	sDate := WORD_TO_STRING(TimeStruct.wYear);
	sDate := CONCAT(sDate,'-');
	IF TimeStruct.wMonth < 10 THEN sDate := CONCAT(sDate, '0');	END_IF
	sDate := CONCAT(sDate,WORD_TO_STRING(TimeStruct.wMonth));
	sDate := CONCAT(sDate,'-');
	IF TimeStruct.wDay < 10 THEN sDate := CONCAT(sDate, '0');	END_IF
	sDate := CONCAT(sDate,WORD_TO_STRING(TimeStruct.wDay));
	
	sTime := '';
	IF TimeStruct.wHour < 10 THEN sTime := CONCAT(sTime, '0');	END_IF
	sTime := CONCAT(sTime, WORD_TO_STRING(TimeStruct.wHour));
	sTime := CONCAT(sTime,':');
	IF TimeStruct.wMinute < 10 THEN sTime := CONCAT(sTime, '0');END_IF
	sTime := CONCAT(sTime,WORD_TO_STRING(TimeStruct.wMinute));
	sTime := CONCAT(sTime,':');
	IF TimeStruct.wSecond < 10 THEN sTime := CONCAT(sTime, '0');END_IF
	sTime := CONCAT(sTime,WORD_TO_STRING(TimeStruct.wSecond)); 
	sTime := CONCAT(sTime,'.');
	IF TimeStruct.wMilliseconds < 100 THEN sTime := CONCAT(sTime, '0');END_IF
	IF TimeStruct.wMilliseconds <  10 THEN sTime := CONCAT(sTime, '0');END_IF
	sTime := CONCAT(sTime,WORD_TO_STRING(TimeStruct.wMilliseconds)); 




IF NOT ((stCommand.eCommandType = eMoverCommand_eGearOutOfSync) OR (stCommand.eCommandType = eMoverCommand_eGearInInSync)) THEN
	THIS^.stLastCommand := stCommand;
END_IF



stMoverAxisCommand := stMoverAxisCommandClear;
CASE _eLogSeverity OF
	
	TcEventSeverity.Critical :;
	
	TcEventSeverity.ERROR:;
	
	TcEventSeverity.INFO:;
	
	TcEventSeverity.VERBOSE:
		
		CASE stCommand.eCommandType OF	

		eMoverCommand_eSetPosition:
			fbFormatString.sFormat := 'SetPosition: X:%.1f;Y:%.1f;C:%.1f';
			fbFormatString.arg1    := F_LREAL(stCommand.stSetPosition.fPositionX);
			fbFormatString.arg2    := F_LREAL(stCommand.stSetPosition.fPositionY);
			fbFormatString.arg3    := F_LREAL(stCommand.stSetPosition.fPositionC);		
			fbFormatString();				
			stMoverAxisCommand.sCommandType   := MoverCommandToString(stCommand.eCommandType);
			stMoverAxisCommand.sTimeStamp 	  := stCommand.stTimeStamp;
			stMoverAxisCommand.sTimeStampDate := sDate;
			stMoverAxisCommand.sTimeStampTime := sTime;
			stMoverAxisCommand.sStation       := stCommand.sText;
			stMoverAxisCommand.sText      	  := fbFormatString.sOut;
				
		eMoverCommand_eReset:
			stMoverAxisCommand.sCommandType   := MoverCommandToString(stCommand.eCommandType);
			stMoverAxisCommand.sTimeStamp 	  := stCommand.stTimeStamp;
			stMoverAxisCommand.sTimeStampDate := sDate;
			stMoverAxisCommand.sTimeStampTime := sTime;
			stMoverAxisCommand.sStation       := stCommand.sText;
			stMoverAxisCommand.sText      	  := 'Reset Cmd';		
	
		eMoverCommand_eEnable:
			stMoverAxisCommand.sCommandType   := MoverCommandToString(stCommand.eCommandType);
			stMoverAxisCommand.sTimeStamp 	  := stCommand.stTimeStamp;
			stMoverAxisCommand.sTimeStampDate := sDate;
			stMoverAxisCommand.sTimeStampTime := sTime;
			stMoverAxisCommand.sStation       := stCommand.sText;
			stMoverAxisCommand.sText      	  := 'Enable Cmd';

		eMoverCommand_eDisable:			
			stMoverAxisCommand.sCommandType   := MoverCommandToString(stCommand.eCommandType);
			stMoverAxisCommand.sStation       := stCommand.sStation;
			stMoverAxisCommand.sText          := 'Disable Cmd';
			stMoverAxisCommand.sTimeStamp 	  := stCommand.stTimeStamp;
			stMoverAxisCommand.sTimeStampDate := sDate;
			stMoverAxisCommand.sTimeStampTime := sTime;

		eMoverCommand_eMoveToPosition:
			fbFormatString.sFormat := 'TargetPos: X:%.1f;Y:%.1f;C:%.1f;Velo:%.2f;Acc:%.0f;Dec:%.0f;Jerk:%.0f';
			fbFormatString.arg1    := F_LREAL(stCommand.stMoveToPositionXYC.fTargetPositionX);
			fbFormatString.arg2    := F_LREAL(stCommand.stMoveToPositionXYC.fTargetPositionY);
			fbFormatString.arg3    := F_LREAL(stCommand.stMoveToPositionXYC.fTargetPositionC);	
			fbFormatString.arg4    := F_LREAL(stCommand.stMoveToPositionXYC.fVelo );	
			fbFormatString.arg5    := F_LREAL(stCommand.stMoveToPositionXYC.fAcc );	
			fbFormatString.arg6    := F_LREAL(stCommand.stMoveToPositionXYC.fDec );
			fbFormatString.arg7    := F_LREAL(stCommand.stMoveToPositionXYC.fJerk );	
			fbFormatString();		
			stMoverAxisCommand.sCommandType   := MoverCommandToString(stCommand.eCommandType);
			stMoverAxisCommand.sStation       := stCommand.sText;	
			stMoverAxisCommand.sText          := fbFormatString.sOut;
			stMoverAxisCommand.sTimeStamp     := stCommand.stTimeStamp;
			stMoverAxisCommand.sTimeStampDate := sDate;
			stMoverAxisCommand.sTimeStampTime := sTime;			

		eMoverCommand_eMoveToPositionXYC:
			fbFormatString.sFormat := 'TargetPos: X:%.1f;Y:%.1f;C:%.1f;Velo:%.2f;Acc:%.0f;Dec:%.0f;Jerk:%.0f';
			fbFormatString.arg1    := F_LREAL(stCommand.stMoveToPositionXYC.fTargetPositionX);
			fbFormatString.arg2    := F_LREAL(stCommand.stMoveToPositionXYC.fTargetPositionY);
			fbFormatString.arg3    := F_LREAL(stCommand.stMoveToPositionXYC.fTargetPositionC);	
			fbFormatString.arg4    := F_LREAL(stCommand.stMoveToPositionXYC.fVelo );	
			fbFormatString.arg5    := F_LREAL(stCommand.stMoveToPositionXYC.fAcc );	
			fbFormatString.arg6    := F_LREAL(stCommand.stMoveToPositionXYC.fDec );
			fbFormatString.arg7    := F_LREAL(stCommand.stMoveToPositionXYC.fJerk );	
			fbFormatString();		
			stMoverAxisCommand.sCommandType   := MoverCommandToString(stCommand.eCommandType);
			stMoverAxisCommand.sStation       := stCommand.sText;	
			stMoverAxisCommand.sText          := fbFormatString.sOut;
			stMoverAxisCommand.sTimeStamp     := stCommand.stTimeStamp;
			stMoverAxisCommand.sTimeStampDate := sDate;
			stMoverAxisCommand.sTimeStampTime := sTime;	

		eMoverCommand_eMoveToPositionExt:
			fbFormatString.sFormat := 'XargetPos: X:%.1f;Y:%.1f;C:%.1f;V:%.2f;A:%.0f;D:%.0f;J:%.0f';
			fbFormatString.arg1    := F_LREAL(stCommand.stMoveToPositionExt.fTargetPositionX);
			fbFormatString.arg2    := F_LREAL(stCommand.stMoveToPositionExt.fTargetPositionY);
			fbFormatString.arg3    := F_LREAL(stCommand.stMoveToPositionExt.fTargetPositionC);	
			fbFormatString.arg4    := F_LREAL(stCommand.stMoveToPositionExt.fVelo );	
			fbFormatString.arg5    := F_LREAL(stCommand.stMoveToPositionExt.fAcc );	
			fbFormatString.arg6    := F_LREAL(stCommand.stMoveToPositionExt.fDec );
			fbFormatString.arg7    := F_LREAL(stCommand.stMoveToPositionExt.fJerk );	
			
			fbFormatString();	
			tempString06 := fbFormatString.sOut;			
			IF stCommand.stMoveToPositionExt.stMoveToPositionOptions.useOrientation THEN
				tempString06 := CONCAT(tempString06,' Or:T');
			ELSE
				tempString06 := CONCAT(tempString06,' Or:F');
			END_IF
					
				
			stMoverAxisCommand.sCommandType   := MoverCommandToString(stCommand.eCommandType);
			stMoverAxisCommand.sStation       := stCommand.sText;	
			stMoverAxisCommand.sText          := tempString06;
			stMoverAxisCommand.sTimeStamp     := stCommand.stTimeStamp;
			stMoverAxisCommand.sTimeStampDate := sDate;
			stMoverAxisCommand.sTimeStampTime := sTime;	


			
		eMoverCommand_eMoveA:
			stMoverAxisCommand.sCommandType   := MoverCommandToString(stCommand.eCommandType);
			stMoverAxisCommand.sStation 	  := stCommand.sStation;
			fbFormatString.sFormat	 		  := 'Position: %.2f; Vel %.0f; acc %.0f; Dec %.0f; Jerk %.0f;   '; 
			fbFormatString.arg1 			  := F_LREAL(stCommand.stMoveOnTrackParameter.fTargetPosition);
			fbFormatString.arg2 			  := F_LREAL(stCommand.stMoveOnTrackParameter.fVelo);
			fbFormatString.arg3 			  := F_LREAL(stCommand.stMoveOnTrackParameter.fAcc);
			fbFormatString.arg4 			  := F_LREAL(stCommand.stMoveOnTrackParameter.fDec);
			fbFormatString.arg5 			  := F_LREAL(stCommand.stMoveOnTrackParameter.fJerk);
			fbFormatString();
			stMoverAxisCommand.sText 		  := fbFormatString.sOut;
			stMoverAxisCommand.sTimeStamp 	  := stCommand.stTimeStamp;
			stMoverAxisCommand.sTimeStampDate := sDate;
			stMoverAxisCommand.sTimeStampTime := sTime;	
	
		eMoverCommand_eMoveB:
			stMoverAxisCommand.sCommandType   := MoverCommandToString(stCommand.eCommandType);
			stMoverAxisCommand.sStation 	  := stCommand.sStation;
			fbFormatString.sFormat	 		  := 'Position: %.2f; Vel %.0f; acc %.0f; Dec %.0f; Jerk %.0f;   '; 
			fbFormatString.arg1 			  := F_LREAL(stCommand.stMoveOnTrackParameter.fTargetPosition);
			fbFormatString.arg2 			  := F_LREAL(stCommand.stMoveOnTrackParameter.fVelo);
			fbFormatString.arg3 			  := F_LREAL(stCommand.stMoveOnTrackParameter.fAcc);
			fbFormatString.arg4 			  := F_LREAL(stCommand.stMoveOnTrackParameter.fDec);
			fbFormatString.arg5 			  := F_LREAL(stCommand.stMoveOnTrackParameter.fJerk);
			fbFormatString();
			stMoverAxisCommand.sText 		  := fbFormatString.sOut;
			stMoverAxisCommand.sTimeStamp 	  := stCommand.stTimeStamp;
			stMoverAxisCommand.sTimeStampDate := sDate;
			stMoverAxisCommand.sTimeStampTime := sTime;	

		eMoverCommand_eMoveC:
			stMoverAxisCommand.sCommandType   := MoverCommandToString(stCommand.eCommandType);
			stMoverAxisCommand.sStation 	  := stCommand.sStation;
			fbFormatString.sFormat	 		  := 'Position: %.2f; Vel %.0f; acc %.0f; Dec %.0f; Jerk %.0f;   '; 
			fbFormatString.arg1 			  := F_LREAL(stCommand.stMoveOnTrackParameter.fTargetPosition);
			fbFormatString.arg2 			  := F_LREAL(stCommand.stMoveOnTrackParameter.fVelo);
			fbFormatString.arg3 			  := F_LREAL(stCommand.stMoveOnTrackParameter.fAcc);
			fbFormatString.arg4 			  := F_LREAL(stCommand.stMoveOnTrackParameter.fDec);
			fbFormatString.arg5 			  := F_LREAL(stCommand.stMoveOnTrackParameter.fJerk);
			fbFormatString();
			stMoverAxisCommand.sText 		  := fbFormatString.sOut;
			stMoverAxisCommand.sTimeStamp 	  := stCommand.stTimeStamp;
			stMoverAxisCommand.sTimeStampDate := sDate;
			stMoverAxisCommand.sTimeStampTime := sTime;				
					
		eMoverCommand_eMoveZ:
			stMoverAxisCommand.sCommandType   := MoverCommandToString(stCommand.eCommandType);
			fbFormatString.sFormat	 		  := 'Position: %.2f; Vel %.0f; acc %.0f; Dec %.0f; Jerk %.0f;   '; 
			fbFormatString.arg1 			  := F_LREAL(stCommand.stMoveOnTrackParameter.fTargetPosition);
			fbFormatString.arg2 			  := F_LREAL(stCommand.stMoveOnTrackParameter.fVelo);
			fbFormatString.arg3 			  := F_LREAL(stCommand.stMoveOnTrackParameter.fAcc);
			fbFormatString.arg4 			  := F_LREAL(stCommand.stMoveOnTrackParameter.fDec);
			fbFormatString.arg5 			  := F_LREAL(stCommand.stMoveOnTrackParameter.fJerk);
			fbFormatString();
			stMoverAxisCommand.sText 		  := fbFormatString.sOut;
			stMoverAxisCommand.sStation 	  := stCommand.sStation;
			stMoverAxisCommand.sTimeStamp 	  := stCommand.stTimeStamp;
			stMoverAxisCommand.sTimeStampDate := sDate;
			stMoverAxisCommand.sTimeStampTime := sTime;	
			
		eMoverCommand_eJoinTrack:
			stMoverAxisCommand.sCommandType   := MoverCommandToString(stCommand.eCommandType);
			fbFormatString.sFormat            := 'TrackOID: %d; Vel %.0f; acc %.0f; Jerk %.0f; ';
			fbFormatString.arg1               := F_UDINT(stCommand.stJoinTrackParameter.nTargetTrack);
			fbFormatString.arg2				  := F_LREAL(stCommand.stJoinTrackParameter.fVelo); 
			fbFormatString.arg3				  := F_LREAL(stCommand.stJoinTrackParameter.fAcc); 
			fbFormatString.arg4				  := F_LREAL(stCommand.stJoinTrackParameter.fJerk); 
			fbFormatString();
			stMoverAxisCommand.sText          := fbFormatString.sOut;	
			stMoverAxisCommand.sStation 	  := stCommand.sStation;
			stMoverAxisCommand.sTimeStamp 	  := stCommand.stTimeStamp;		
			stMoverAxisCommand.sTimeStampDate := sDate;
			stMoverAxisCommand.sTimeStampTime := sTime;			
			
		eMoverCommand_eLeaveTrack:
			stMoverAxisCommand.sCommandType   := MoverCommandToString(stCommand.eCommandType);
			fbFormatString.sFormat            := 'Pos: X:%.1f; Y:%.1f; C:%.1f; Vel:%.0f  Acc:%.0f; Dec:%.0f Jerk %.0f';
			fbFormatString.arg1               := F_LREAL(stCommand.stLeaveTrackParameter.fPositionX);
			fbFormatString.arg2               := F_LREAL(stCommand.stLeaveTrackParameter.fPositionY);
			fbFormatString.arg3               := F_LREAL(stCommand.stLeaveTrackParameter.fPositionC);
			fbFormatString.arg4				  := F_LREAL(stCommand.stLeaveTrackParameter.fVelo); 
			fbFormatString.arg5				  := F_LREAL(stCommand.stLeaveTrackParameter.fAcc); 
			fbFormatString.arg6				  := F_LREAL(stCommand.stLeaveTrackParameter.fDec); 
			fbFormatString.arg7				  := F_LREAL(stCommand.stLeaveTrackParameter.fJerk); 
			fbFormatString();
			stMoverAxisCommand.sText          := fbFormatString.sOut;	
			stMoverAxisCommand.sStation 	  := stCommand.sStation;
			stMoverAxisCommand.sTimeStamp 	  := stCommand.stTimeStamp;		
			stMoverAxisCommand.sTimeStampDate := sDate;
			stMoverAxisCommand.sTimeStampTime := sTime;			
	

		eMoverCommand_eLeaveTrackInPosition:
			stMoverAxisCommand.sCommandType   := MoverCommandToString(stCommand.eCommandType);
			fbFormatString.sFormat            := 'Pos: X:%.1f; Y:%.1f; C:%.1f';
			fbFormatString.arg1               := F_LREAL(stCommand.stLeaveTrackInPositionParameter.fPositionX);
			fbFormatString.arg2               := F_LREAL(stCommand.stLeaveTrackInPositionParameter.fPositionY);
			fbFormatString.arg3               := F_LREAL(stCommand.stLeaveTrackInPositionParameter.fPositionC);
			fbFormatString();
			stMoverAxisCommand.sText          := fbFormatString.sOut;	
			stMoverAxisCommand.sStation 	  := stCommand.sStation;
			stMoverAxisCommand.sTimeStamp 	  := stCommand.stTimeStamp;		
			stMoverAxisCommand.sTimeStampDate := sDate;
			stMoverAxisCommand.sTimeStampTime := sTime;			

		eMoverCommand_eMoveModOnTrack:
			fbFormatString.sFormat := 'TargetPos:%.4f;Velo:%.2f;Acc:%.0f;Jerk:%.0f;Gap:%.0f;TargetTrack:%d $n ;ActSetPos:%.2f;ActSetOid:%d;ActVelo:%.0f;ActAcc:%.0f;';
			fbFormatString.arg1 := F_LREAL(stCommand.stMoveOnTrackParameter.fTargetPosition);
			fbFormatString.arg2 := F_LREAL(stCommand.stMoveOnTrackParameter.fVelo );	
			fbFormatString.arg3 := F_LREAL(stCommand.stMoveOnTrackParameter.fAcc );	
			fbFormatString.arg4 := F_LREAL(stCommand.stMoveOnTrackParameter.fJerk );
			fbFormatString.arg5 := F_LREAL(stCommand.stMoveOnTrackParameter.fGap);
			fbFormatString.arg6 := F_UDINT(stCommand.stMoveOnTrackParameter.nTargetTrackOid);
			fbFormatString.arg7 := F_LREAL(stCommand.stActualParameter.fSetTrackPosition);
			fbFormatString.arg8 := F_UDINT(stCommand.stActualParameter.nTrackOid);	
			fbFormatString.arg9 := F_LREAL(stCommand.stActualParameter.fSetVelo);	
			fbFormatString.arg10:= F_LREAL(stCommand.stActualParameter.fSetAcc);			
			fbFormatString();
			
			stMoverAxisCommand.sCommandType   := MoverCommandToString(stCommand.eCommandType);
			stMoverAxisCommand.sStation       := stCommand.sStation;				
			stMoverAxisCommand.sText          := fbFormatString.sOut;
			stMoverAxisCommand.sTimeStamp     := stCommand.stTimeStamp;
			stMoverAxisCommand.sTimeStampDate := sDate;
			stMoverAxisCommand.sTimeStampTime := sTime;
			
		
		eMoverCommand_eGearInPosOnTrack:
				
			fbFormatString.sFormat := 'MaSyncPos:%.4f;SlSyncPos:%.4f;SlSyncDir:%d;SlSyncPosDir:%d;$nSyncTolDist:%.2f;TolSlSyncPos:%.2f,SyncTr:%d,TrailSize:%d$n';
							
			fbFormatString.arg1 := F_LREAL(stCommand.stGearInPosOnTrackParameter.MasterSyncPos);
			fbFormatString.arg2 := F_LREAL(stCommand.stGearInPosOnTrackParameter.SlaveSyncPos);
			fbFormatString.arg3 := F_UINT(stCommand.stGearInPosOnTrackParameter.allowedSlaveSyncDirections);
			fbFormatString.arg4 := F_UINT(stCommand.stGearInPosOnTrackParameter.directionSlaveSyncPosition);
			fbFormatString.arg5 := F_LREAL(stCommand.stGearInPosOnTrackParameter.inSyncToleranceDistance);
			fbFormatString.arg6 := F_LREAL(stCommand.stGearInPosOnTrackParameter.moduloToleranceSlaveSyncPosition);
			fbFormatString.arg7 := F_UDINT(stCommand.stGearInPosOnTrackParameter.Track);
			fbFormatString.arg8 := F_UDINT(stCommand.stGearInPosOnTrackParameter.TrackTrailSize);	
			fbFormatString();
			tempString01 := fbFormatString.sOut;
					
			fbFormatString.sFormat := 'Velo:%.2f;Acc:%.0f;Dec:%.0f;Jerk:%.0f;Gap:%.0f';
			fbFormatString.arg1 := F_LREAL(stCommand.stGearInPosOnTrackParameter.Velocity);
			fbFormatString.arg2 := F_LREAL(stCommand.stGearInPosOnTrackParameter.Acceleration);
			fbFormatString.arg3 := F_LREAL(stCommand.stGearInPosOnTrackParameter.Deceleration);
			fbFormatString.arg4 := F_LREAL(stCommand.stGearInPosOnTrackParameter.Jerk);
			fbFormatString.arg5 := F_LREAL(stCommand.stGearInPosOnTrackParameter.Gap);
			fbFormatString();
			tempString02 := fbFormatString.sOut;
		
			stMoverAxisCommand.sCommandType   := MoverCommandToString(stCommand.eCommandType);
			stMoverAxisCommand.sStation       := stCommand.sStation;				
			stMoverAxisCommand.sText          := CONCAT(tempString01,tempString02);
			stMoverAxisCommand.sTimeStamp     := stCommand.stTimeStamp;
			stMoverAxisCommand.sTimeStampDate := sDate;
			stMoverAxisCommand.sTimeStampTime := sTime;			


			
			
			
		eMoverCommand_eGearInPosOnTrackMasterMover:
				
			fbFormatString.sFormat := 'Ma:%d;MaSyncPos:%.4f;TrMaSP:%d;$n';
			fbFormatString.arg1 := F_UDINT(stCommand.stGearInPosOnTrackMasterMoverParameter.MasterMover);
			fbFormatString.arg2 := F_LREAL(stCommand.stGearInPosOnTrackMasterMoverParameter.MasterSyncPos);
			fbFormatString.arg3 := F_UDINT(stCommand.stGearInPosOnTrackMasterMoverParameter.TrackMasterSyncPos);
			fbFormatString();
			tempString01 := fbFormatString.sOut;
			
			fbFormatString.sFormat :=('SlSyncPos:%.2f;TrSlSP:%d$n');
			fbFormatString.arg1 := F_LREAL(stCommand.stGearInPosOnTrackMasterMoverParameter.SlaveSyncPos);
			fbFormatString.arg2 := F_UDINT(stCommand.stGearInPosOnTrackMasterMoverParameter.TrackSlaveSyncPos);			
			fbFormatString();
			tempString02 := fbFormatString.sOut;				
			
			fbFormatString.sFormat := 'TolMa:%.2f;MaDir:%d;SynTolD:%.2f;TolSlSP:%.2f;SlDir:%d;SlDirSync:%d$n';
			fbFormatString.arg1 := F_LREAL(stCommand.stGearInPosOnTrackMasterMoverParameter.moduloToleranceMasterSyncPosition);
			fbFormatString.arg2 := F_DINT(stCommand.stGearInPosOnTrackMasterMoverParameter.directionMasterSyncPosition);
			fbFormatString.arg3 := F_LREAL(stCommand.stGearInPosOnTrackMasterMoverParameter.inSyncToleranceDistance);
			fbFormatString.arg4 := F_LREAL(stCommand.stGearInPosOnTrackMasterMoverParameter.moduloToleranceSlaveSyncPosition);
			fbFormatString.arg5 := F_DINT(stCommand.stGearInPosOnTrackMasterMoverParameter.allowedSlaveSyncDirections);
			fbFormatString.arg6 := F_DINT(stCommand.stGearInPosOnTrackMasterMoverParameter.directionSlaveSyncPosition);
			fbFormatString();
			tempString03 := fbFormatString.sOut;				
			
			fbFormatString.sFormat := 'Velo:%.2f;Acc:%.0f;Dec:%.0f;Jerk:%.0f;';
			fbFormatString.arg1 := F_LREAL(stCommand.stGearInPosOnTrackMasterMoverParameter.Velocity);
			fbFormatString.arg2 := F_LREAL(stCommand.stGearInPosOnTrackMasterMoverParameter.Acceleration);
			fbFormatString.arg3 := F_LREAL(stCommand.stGearInPosOnTrackMasterMoverParameter.Deceleration);
			fbFormatString.arg4 := F_LREAL(stCommand.stGearInPosOnTrackMasterMoverParameter.Jerk);
			fbFormatString();
			tempString04 := fbFormatString.sOut;
			
			tempString05 := CONCAT(tempString01,tempString02);
			tempString05 := CONCAT(tempString05,tempString03);
			//tempString05 := CONCAT(tempString05,tempString04);
			
			stMoverAxisCommand.sCommandType   := MoverCommandToString(stCommand.eCommandType);
			stMoverAxisCommand.sStation       := stCommand.sStation;				
			stMoverAxisCommand.sText          := tempString05;
			stMoverAxisCommand.sTimeStamp     := stCommand.stTimeStamp;
			stMoverAxisCommand.sTimeStampDate := sDate;
			stMoverAxisCommand.sTimeStampTime := sTime;	



			
		
		eMoverCommand_eHalt:
			//fbResult.SendMessage(Tc_Events.Tc3_XPlanarStandardEventClass.HaltCommand,
			//						TC_EVENT_CLASSES.Tc3_XPlanarStandardEventClass,stCommand,stActualMotionParameter);					
			fbFormatString.sFormat 	:= 'Dec_XY: %.0f; Jerk_XY: %.0f; Dec_C: %.0f; Jerk_C: %.0f  $nPos_XYT: %.3f; %.3f; %.3f; ';
			fbFormatString.arg1    	:= F_LREAL(stCommand.stHaltParameter.fDeceleration_XY);
			fbFormatString.arg2    	:= F_LREAL(stCommand.stHaltParameter.fJerk_XY);				
			fbFormatString.arg3    	:= F_LREAL(stCommand.stHaltParameter.fDeceleration_C);	
			fbFormatString.arg4    	:= F_LREAL(stCommand.stHaltParameter.fJerk_C);
			fbFormatString.arg5  	:= F_LREAL(SetPos.x);
			fbFormatString.arg6 	:= F_LREAL(SetPos.y);
			fbFormatString.arg7 	:= F_LREAL(SetOnTrack.SetPos);
			fbFormatString();			
				
			stMoverAxisCommand.sCommandType   := MoverCommandToString(stCommand.eCommandType);
			stMoverAxisCommand.sStation 	  := stCommand.sStation;				
			stMoverAxisCommand.sText 		  := fbFormatString.sOut;
			stMoverAxisCommand.sTimeStamp 	  := stCommand.stTimeStamp;
			stMoverAxisCommand.sTimeStampDate := sDate;
			stMoverAxisCommand.sTimeStampTime := sTime;
								
		eMoverCommand_eEnableExternalSetPos :	
			stMoverAxisCommand.sCommandType   := MoverCommandToString(stCommand.eCommandType);
			stMoverAxisCommand.sStation 	  := stCommand.sStation;
			stMoverAxisCommand.sTimeStamp 	  := stCommand.stTimeStamp;	
			stMoverAxisCommand.sText 		  := stCommand.sText;
			stMoverAxisCommand.sTimeStampDate := sDate;
			stMoverAxisCommand.sTimeStampTime := sTime;

		eMoverCommand_eAddMoverToGroup :	
			stMoverAxisCommand.sCommandType   := MoverCommandToString(stCommand.eCommandType);
			stMoverAxisCommand.sStation 	  := 'Add Mover to Group';
			stMoverAxisCommand.sTimeStamp 	  := stCommand.stTimeStamp;
			stMoverAxisCommand.sTimeStampDate := sDate;
			stMoverAxisCommand.sTimeStampTime := sTime;		
			stMoverAxisCommand.sText      	  := CONCAT('GrupOID: ', stCommand.sText);

		eMoverCommand_eRemoveMoverFromGroup :	
			stMoverAxisCommand.sCommandType   := MoverCommandToString(stCommand.eCommandType);
			stMoverAxisCommand.sStation 	  := 'Remove mover from Group';
			stMoverAxisCommand.sTimeStamp 	  := stCommand.stTimeStamp;
			stMoverAxisCommand.sTimeStampDate := sDate;
			stMoverAxisCommand.sTimeStampTime := sTime;		
			stMoverAxisCommand.sText      	  := 'Remove Mover from Group Cmd';				
						
		END_CASE
		
	TcEventSeverity.WARNING:;

END_CASE



aLog[0] :=  stMoverAxisCommand;
FOR nCntBuffer := UINT_TO_INT(MAX_LAST_LOGS) TO 1  BY -1 DO
	MEMCPY(destAddr:=ADR(aLog[nCntBuffer]) , srcAddr:=ADR(aLog[nCntBuffer-1]) , n:=SIZEOF(ST_MoverCommandLog) );
	aLog[nCntBuffer].nNo := nCntBuffer;
	MEMSET(destAddr:=ADR(aLog[nCntBuffer-1]) , fillByte:=0 , n:= SIZEOF(ST_MoverCommandLog));
END_FOR
END_METHOD



METHOD CheckStartConditions : ST_CheckStartConditionFeedback


VAR_INST
	
	CurrentPosition				: MoverVector;
	
	fCurrentPositionX			: LREAL;
	fCurrentPositionX_Temp		: LREAL;
	fDividerX					: LREAL;
	
	fCurrentPositionY			: LREAL;
	fCurrentPositionY_Temp		: LREAL;
	fDividerY					: LREAL;

	fCurrentAngleC				: LREAL;
	fCurrentAngleC_Temp			: LREAL;
	fCurrentAngleC_Deviation	: LREAL;
	fDividerC					: LREAL;
	
	bPositionXLimitExceeded		: BOOL;
	bPositionYLimitExceeded		: BOOL;
	bAngleLimitExceeded			: BOOL;
	bCheckStartConditions		: BOOL;
	fCurrentPositionX_Deviation	: LREAL;
	fCurrentPositionY_Deviation	: LREAL;
	bAngleLimitExceededResult	: BOOL;
	
END_VAR

	  CurrentPosition := stMoverRef.MCTOPLC.ACT.ActPos;
	fCurrentPositionX := ABS(CurrentPosition.x);
	fCurrentPositionY := ABS(CurrentPosition.y);
	   fCurrentAngleC := ABS(CurrentPosition.c);
	


	// Angle-Limit
	IF fCurrentAngleC > 90.0
	OR fCurrentAngleC < 90.0
	THEN
		fDividerC := LTRUNC(fCurrentAngleC/90.0);
	ELSE
		fDividerC := 0;
	END_IF		
	fCurrentAngleC_Temp := fCurrentAngleC - fDividerC * 90.0;
	
	IF fCurrentAngleC_Temp > 45.0 THEN
		fCurrentAngleC_Deviation := fCurrentAngleC_Temp - 90.0;
	ELSIF fCurrentAngleC_Temp < -45.0 THEN
		fCurrentAngleC_Deviation := fCurrentAngleC_Temp + 90.0;
	ELSE
		fCurrentAngleC_Deviation := fCurrentAngleC_Temp;
	END_IF	
	
	IF ABS(fCurrentAngleC_Deviation) > 10.0 THEN
		bAngleLimitExceeded := TRUE;
	ELSE
		bAngleLimitExceeded := FALSE;
	END_IF
	
	

	// Position X-Limit
	IF fCurrentPositionX < 120.0
	OR fCurrentPositionX > 120.0
	THEN
		fDividerX := LTRUNC(fCurrentPositionX/120.0);
	ELSE
		fDividerX := 0;
	END_IF
	fCurrentPositionX_Temp := fCurrentPositionX - fDividerX * 120.0;

	IF fCurrentPositionX_Temp > 60.0 THEN
		fCurrentPositionX_Deviation := fCurrentPositionX_Temp - 120;
	ELSIF fCurrentPositionX_Temp < -60.0 THEN
		fCurrentPositionX_Deviation := fCurrentPositionX_Temp + 120;
	ELSE
		fCurrentPositionX_Deviation := fCurrentPositionX_Temp;
	END_IF

	IF ABS(fCurrentPositionX_Deviation) > 1.0 THEN
		bPositionXLimitExceeded := TRUE;
	ELSE
		bPositionXLimitExceeded := FALSE;
	END_IF
	
	
		
	// Position Y-Limit
	IF fCurrentPositionY < 120.0
	OR fCurrentPositionY > 120.0
	THEN
		fDividerY := LTRUNC(fCurrentPositionY/120.0);
	ELSE
		fDividerY := 0;
	END_IF
	fCurrentPositionY_Temp := fCurrentPositionY - fDividerY * 120.0;

	IF fCurrentPositionY_Temp > 60.0 THEN
		fCurrentPositionY_Deviation := fCurrentPositionY_Temp - 120;
	ELSIF fCurrentPositionY_Temp < -60.0 THEN
		fCurrentPositionY_Deviation := fCurrentPositionY_Temp + 120;
	ELSE
		fCurrentPositionY_Deviation := fCurrentPositionY_Temp;
	END_IF

	IF ABS(fCurrentPositionY_Deviation) > 1.0 THEN
		bPositionYLimitExceeded := TRUE;
	ELSE
		bPositionYLimitExceeded := FALSE;
	END_IF	
	
	
		
	// Checking angle limit depending on position limit
	IF  bAngleLimitExceeded 
	AND (bPositionXLimitExceeded OR  bPositionYLimitExceeded)
	THEN
		bAngleLimitExceededResult := TRUE;
		    bCheckStartConditions := FALSE;
	ELSE
		bAngleLimitExceededResult := FALSE;
		    bCheckStartConditions := TRUE;
	END_IF
	
	

	// Result
	CheckStartConditions.nMoverID			   	 	 := nId;
	CheckStartConditions.bPositionOK             	 := bCheckStartConditions;
	CheckStartConditions.bAngleLimitExceeded     	 := bAngleLimitExceededResult;
	CheckStartConditions.bPositionXLimitExceeded 	 := bPositionXLimitExceeded;
	CheckStartConditions.bPositionYLimitExceeded 	 := bPositionYLimitExceeded;	
 	CheckStartConditions.fCurrentAngleDeviation	 	 := fCurrentAngleC_Deviation;
	CheckStartConditions.fCurrentPositionDeviationX  := fCurrentPositionX_Deviation;
	CheckStartConditions.fCurrentPositionDeviationY  := fCurrentPositionY_Deviation;
END_METHOD

METHOD GetCustomTrackID : DINT
VAR_INPUT
END_VAR



VAR_INST
	
	idx					: UDINT;
	nCycleCounterMem	: UDINT;
	GetCustomTrackIdMem	: DINT;
	TrackOidMem			: OTCID;

END_VAR


	IF                nCycleCounter <> nCycleCounterMem
	AND THIS^.P_SetOnTrack.TrackOID <> TrackOidMem
	THEN
		nCycleCounterMem := nCycleCounter;

		IF THIS^.P_SetOnTrack.TrackOID = 0 THEN
			GetCustomTrackID := -1;  // -1: Mover is not on a track
		ELSE
			GetCustomTrackID := -2; // -2: Track not found 
		
			FOR idx:=1 TO Params_XPlanar.maxTrackCount DO 		
				IF CustomTrackIdTable[idx].TrackOID = THIS^.P_SetOnTrack.TrackOID THEN
					   GetCustomTrackID := UDINT_TO_DINT(CustomTrackIdTable[idx].nCustomID);
					GetCustomTrackIdMem := GetCustomTrackId;
					EXIT;
				END_IF
			END_FOR
		END_IF
		TrackOidMem := THIS^.P_SetOnTrack.TrackOID;
	ELSE
		GetCustomTrackID := GetCustomTrackIdMem;
	END_IF
END_METHOD

METHOD GetDistanceToTrack : LREAL    // -1 if track is not enabled

VAR_INPUT
	ipTrack	: I_TrackStandard;
END_VAR
	

VAR_INST
	idx						: ULINT;
	nSteps					: ULINT;
	currentMoverPositon 	: MoverVector;
	fTrackLength			: LREAL;
	positionXYC				: PositionXYC;
	fDistance				: LREAL;
END_VAR



	IF ipTrack.P_State <> MC_PLANAR_STATE.Enabled THEN
		GetDistanceToTrack := -1.0;
	ELSIF stMoverRef.MCTOPLC.SETONTRACK.TrackOID = ipTrack.P_OID THEN
		GetDistanceToTrack := 0.0;
	ELSE	
		currentMoverPositon := stMoverRef.MCTOPLC.ACT.ActPos;
			   fTrackLength := ipTrack.GetLength();
		
		nSteps := LREAL_TO_ULINT(fTrackLength);
		
		FOR idx:=0 TO nSteps DO
			ipTrack.GetMoverPositionAt(MIN(ULINT_TO_LREAL(idx), fTrackLength), positionXYC);
			IF(idx=0) THEN
				fDistance := SQRT(EXPT(ABS(positionXYC.x - currentMoverPositon.x), 2) + EXPT(ABS(positionXYC.y - currentMoverPositon.y), 2));;
			ELSE
				fDistance := MIN(SQRT(EXPT(ABS(positionXYC.x - currentMoverPositon.x), 2) + EXPT(ABS(positionXYC.y - currentMoverPositon.y), 2)), fDistance);	
			END_IF		
		END_FOR
				
		GetDistanceToTrack := fDistance;
	END_IF
END_METHOD

METHOD GetLastKnownCustomTrackID : DINT
VAR_INPUT
END_VAR



VAR_INST
	
	idx					: UDINT;
	nCycleCounterMem	: UDINT;
	GetCustomTrackIdMem	: DINT;
	TrackOidMem			: OTCID;

END_VAR


	GetLastKnownCustomTrackID := -1; // -1: Mover has no track history
	IF nLastKnownTrackOID > 0 THEN
		FOR idx:=1 TO Params_XPlanar.maxTrackCount DO 		
			IF CustomTrackIdTable[idx].TrackOID = nLastKnownTrackOID THEN
				GetLastKnownCustomTrackID := UDINT_TO_DINT(CustomTrackIdTable[idx].nCustomID);
				EXIT;
			END_IF
		END_FOR
	END_IF
END_METHOD

METHOD MoveOnTrack : BOOL
VAR_INPUT
	sLogMessage			: STRING;
	ipTrack				: I_TrackStandard;
	trackPosition       : LREAL;
	velocity           	: LREAL;
	acceleration        : LREAL;
	jerk                : LREAL;
	gap					: LREAL;
	direction			: Tc3_Mc3PlanarMotion.MC_DIRECTION := Tc3_Mc3PlanarMotion.MC_DIRECTION.mcDirectionPositive;
END_VAR

VAR_INST 
	dyn : DynamicConstraint_PathXY;	 
END_VAR
	
VAR
	stMoveOnTrackOptions	: ST_MoveOnTrackOptions;

	stCommand 			: ST_MoverCommand; 
	fAbsolutePositon 	: LREAL; // 
	xCommandMissed		: BOOL;
	ref 				: POINTER TO MC_PlanarTrack; 
	//stOptions			: ST_MoveAbsoluteCAOptions; 
END_VAR

VAR_INST
	_ipTrack			: I_TrackStandard;
	_trackPosition      : LREAL;
	_velocity           : LREAL;
	_acceleration       : LREAL;
	_jerk               : LREAL;
	_gap				: LREAL;
	_ref				: POINTER TO MC_PlanarTrack; 
	
	idx					: UDINT;
	nTrackID			: UDINT;
	

END_VAR
MEMSET(ADR(stRtMoveOnTrack), 0, SIZEOF(stRtMoveOnTrack));

ref := ipTrack.ref;

_ref				:= ref;
_trackPosition      := trackPosition;
_velocity           := velocity;
_acceleration       := acceleration;
_jerk               := jerk;
_gap				:= gap;


dyn.SetValuesVADJ(velocity,acceleration, acceleration, jerk); 
stMoveOnTrackOptions.direction := direction;
stMoveOnTrackOptions.gap       := gap;
stMoverRef.MoveOnTrack(moveOnTrackCmdFB, ref^, trackPosition, dyn, stMoveOnTrackOptions);


// Store the command parameters for retriggering the command later on.
stMoveOnTrackParameter.fTrackPosition	:= trackPosition;
stMoveOnTrackParameter.fVelo			:= velocity;
stMoveOnTrackParameter.ipTrack			:= ipTrack;
stMoveOnTrackParameter.fAcc				:= acceleration;
stMoveOnTrackParameter.fDec				:= acceleration;
stMoveOnTrackParameter.fJerk			:= jerk;
stMoveOnTrackParameter.fGap				:= gap;
stMoveOnTrackParameter.direction		:= direction;


// Command History
stCommand.eCommandType                           := eMoverCommand_eMoveModOnTrack;
stCommand.sStation                               := sLogMessage;
stCommand.stMoveOnTrackParameter.fTargetPosition := trackPosition ;
stCommand.stMoveOnTrackParameter.nTargetTrackOid := ref^.MCTOPLC_STD.TrackOID;
stCommand.stMoveOnTrackParameter.nTargetTrackID  := nTrackID;
stCommand.stMoveOnTrackParameter.fAcc 	         := acceleration;
stCommand.stMoveOnTrackParameter.fDec 	         := acceleration;
stCommand.stMoveOnTrackParameter.fJerk 	         := jerk;
stCommand.stMoveOnTrackParameter.fVelo 	         := velocity;
stCommand.stMoveOnTrackParameter.fGap 	         := gap;
stCommand.stActualParameter 			         := UpdateActualMotionParameter();
UpdateCommandHistory(stCommand);


MoveOnTrack := TRUE;
END_METHOD


{attribute 'obsolete' := 'Obsolete: Please use MoveToPositionExt instead'}
METHOD MoveToPosition  : BOOL
VAR_INPUT
	slogMessage		: STRING;
	targetPosition	: REFERENCE TO PositionXYC;
	velocity		: LREAL;
	acceleration	: LREAL;
	deceleration	: LREAL;
	jerk			: LREAL;
END_VAR

VAR_INST
	DynamicConstraintPath : DynamicConstraint_PathXY;   
END_VAR
			
VAR
	stMoveToPositionOptions		: ST_MoveToPositionOptions;
	stCommand 					: ST_MoverCommand;
END_VAR
MEMSET(ADR(stRtMoveToPos), 0, SIZEOF(stRtMoveToPos));
DynamicConstraintPath.SetValuesVADJ(velocity,acceleration,deceleration,jerk);

stMoveToPositionOptions.useOrientation := FALSE;
stMoverRef.MoveToPosition(moveToPosCmdFB, targetPosition,  DynamicConstraintPath, stMoveToPositionOptions);



// Command History
stCommand.eCommandType 							:= eMoverCommand_eMoveToPosition;
stCommand.sText        							:= slogMessage;
stCommand.stMoveToPosition.fTargetPositionX 	:= targetPosition.x;
stCommand.stMoveToPosition.fTargetPositionY 	:= targetPosition.y;
stCommand.stMoveToPosition.fTargetPositionC 	:= targetPosition.c;
stCommand.stMoveToPosition.fVelo				:= DynamicConstraintPath.V;
stCommand.stMoveToPosition.fAcc 				:= DynamicConstraintPath.A;
stCommand.stMoveToPosition.fDec 				:= DynamicConstraintPath.D;
stCommand.stMoveToPosition.fJerk 				:= DynamicConstraintPath.J;
UpdateCommandHistory(stCommand);



MoveToPosition := TRUE;
END_METHOD

METHOD AddToGroup : BOOL
VAR_INPUT
	group : REFERENCE TO MC_PlanarGroup;
END_VAR


VAR
	stCommand : ST_MoverCommand;
END_VAR
MEMSET(ADR(stRtAddMover), 0, SIZEOF(stRtAddMover));
stMoverRef.AddToGroup(addMoverCmdFB, group);
AddToGroup := TRUE;



// Command History
stCommand.eCommandType 	:= eMoverCommand_eAddMoverToGroup;
stCommand.sText     	:= UDINT_TO_STRING(group.MCTOPLC_STD.GroupOID);
UpdateCommandHistory(stCommand);
END_METHOD

METHOD AdoptTrackOrientation : BOOL
VAR_INPUT
	slogMessage		: STRING;
	velocity		: LREAL;
	acceleration	: LREAL;
	deceleration	: LREAL;
	jerk			: LREAL;
	stOptions 		: REFERENCE TO ST_AdoptTrackOrientationOptions;
END_VAR

VAR_INST
	dyn					 		: DynamicConstraint_Coordinates;
END_VAR

VAR	
	stCommand 					: ST_MoverCommand;
END_VAR
MEMSET(ADR(stRtAdoptTrackOri), 0, SIZEOF(stRtAdoptTrackOri));
dyn.AddLimit(Coord_Mcs_C1,velocity, acceleration, deceleration, jerk);
stMoverRef.AdoptTrackOrientation(adoptTrackOriCmdFB, dyn, stOptions);


// Command History
stCommand.eCommandType 								:= eMoverCommand_eAdoptTrackOrientation;
stCommand.sStation 									:= slogMessage;
stCommand.stMoveOnTrackParameter.fVelo 				:= velocity;
stCommand.stMoveOnTrackParameter.fAcc 				:= acceleration;
stCommand.stMoveOnTrackParameter.fDec 				:= deceleration;
stCommand.stMoveOnTrackParameter.fJerk 				:= jerk;
UpdateCommandHistory(stCommand);
	
AdoptTrackOrientation := TRUE;
END_METHOD

METHOD Disable : BOOL
VAR_INPUT
	sLogMessage: STRING;
END_VAR


VAR
	stCommand : ST_MoverCommand;
END_VAR
MEMSET(ADR(stRtDisable), 0, SIZEOF(stRtDisable));
stMoverRef.Disable(disableCmdFB);

bIsSetpointGeneratorActive := FALSE;

// Command History
stCommand.eCommandType 	:= eMoverCommand_eDisable;
stCommand.sStation     	:= sLogMessage;
UpdateCommandHistory(stCommand);


Disable := TRUE;
END_METHOD

METHOD DisableExternalSetpointGeneration : BOOL
VAR_INPUT
	slogMessage : STRING;
END_VAR


VAR
	stOptions : ST_ExternalSetpointGenerationOptions;
	stCommand : ST_MoverCommand;
END_VAR
MEMSET(ADR(stRtDisableSetPos), 0, SIZEOF(stRtDisableSetPos));
stMoverRef.StopExternalSetpointGeneration(disableExtSetPosCmdFB);
DisableExternalSetpointGeneration := TRUE;

bIsSetpointGeneratorActive := FALSE;

// Command History
stCommand.eCommandType 	:= eMoverCommand_eDisableExternalSetPos;
stCommand.sStation 		:= slogMessage;
UpdateCommandHistory(stCommand);
END_METHOD

METHOD Enable : BOOL
VAR_INPUT
	slogMessage : STRING;
END_VAR

VAR
	stCommand : ST_MoverCommand;
END_VAR
MEMSET(ADR(stRtEnable), 0, SIZEOF(stRtEnable));
stMoverRef.Enable(enableCmdFB);
Enable := TRUE;

// Command History
stCommand.eCommandType 	:= eMoverCommand_eEnable;
stCommand.sText     	:= sLogMessage;

UpdateCommandHistory(stCommand);
END_METHOD

METHOD EnableExternalSetpointGeneration : BOOL
VAR_INPUT
	slogMessage 	: STRING;
	eSetpointMode 	: MC_EXTERNAL_SET_POSITION_MODE;
END_VAR


VAR
	stOptions 	: ST_ExternalSetpointGenerationOptions;
	stCommand 	: ST_MoverCommand;
	sInfoText	: STRING;
END_VAR
MEMSET(ADR(stRtEnableSetPos), 0, SIZEOF(stRtEnableSetPos));

	CASE eSetpointMode OF 
	
	MC_SET_POSITION_MODE.Absolute:
		stOptions.mode := MC_SET_POSITION_MODE.Absolute;
		     sInfoText := 'Mode: Absolute';
		
	MC_SET_POSITION_MODE.Relative:
		stOptions.mode := MC_SET_POSITION_MODE.Relative;
			 sInfoText := 'Mode: Relative';		

	END_CASE


stMoverRef.StartExternalSetpointGeneration(enableExtSetPosCmdFB, stOptions);
EnableExternalSetpointGeneration := TRUE;

bIsSetpointGeneratorActive := TRUE;

// Command History
stCommand.eCommandType 	:= eMoverCommand_eEnableExternalSetPos;
stCommand.sStation 		:= slogMessage;
stCommand.sText  		:= sInfoText;
UpdateCommandHistory(stCommand);
END_METHOD

METHOD GearInPosOnTrack : BOOL
VAR_INPUT
	slogMessage		: STRING;
	master			: OTCID;
	trackTrail		: REFERENCE TO MC_PlanarTrackTrail;
	masterSyncPos	: LREAL;
	slaveSyncPos	: LREAL;
	syncTrack		: I_TrackStandard;
	velocity		: LREAL;
	acceleration	: LREAL;
	deceleration	: LREAL;
	jerk			: LREAL;
	stOptions 		: REFERENCE TO ST_GearInPosOnTrackOptions;
END_VAR


VAR_INST
	dyn					 		: DynamicConstraint_PathXY;	
END_VAR

VAR
	ref							: POINTER TO MC_PlanarTrack;
	stCommand 					: ST_MoverCommand;
END_VAR
	

	MEMSET(ADR(stRtGearInPosOnTrack), 0, SIZEOF(stRtGearInPosOnTrack));
	
	dyn.SetValuesVADJ(velocity, acceleration, deceleration, jerk);
	
	ref := syncTrack.ref;
	stMoverRef.GearInPosOnTrack(gearInPosOnTrackCmdFB, master, trackTrail, masterSyncPos, slaveSyncPos, ref^, dyn, stOptions);
	
	// Command History
	stCommand.eCommandType 								:= eMoverCommand_eGearInPosOnTrack;
	stCommand.sStation 									:= slogMessage;
	
	stCommand.stGearInPosOnTrackParameter.MasterSyncPos := masterSyncPos;
	stCommand.stGearInPosOnTrackParameter.SlaveSyncPos  := slaveSyncPos;
	stCommand.stGearInPosOnTrackParameter.Gap			:= stOptions.gap;
	
	stCommand.stGearInPosOnTrackParameter.Velocity  	:= velocity;
	stCommand.stGearInPosOnTrackParameter.Acceleration  := acceleration;
	stCommand.stGearInPosOnTrackParameter.Deceleration  := deceleration;
	stCommand.stGearInPosOnTrackParameter.Jerk  		:= jerk;
	
	stCommand.stGearInPosOnTrackParameter.allowedSlaveSyncDirections := stOptions.allowedSlaveSyncDirections;
	stCommand.stGearInPosOnTrackParameter.directionSlaveSyncPosition := stOptions.directionSlaveSyncPosition;
	
	stCommand.stGearInPosOnTrackParameter.inSyncToleranceDistance 			:= stOptions.inSyncToleranceDistance;
	stCommand.stGearInPosOnTrackParameter.moduloToleranceSlaveSyncPosition	:= stOptions.moduloToleranceSlaveSyncPosition;
	
	stCommand.stGearInPosOnTrackParameter.Track				:= syncTrack.P_OID;
	
	IF __ISVALIDREF(trackTrail) THEN
		stCommand.stGearInPosOnTrackParameter.TrackTrailSize := trackTrail.Size;
	ELSE
		stCommand.stGearInPosOnTrackParameter.TrackTrailSize := 0;
	END_IF
	
	
	UpdateCommandHistory(stCommand);
		
	GearInPosOnTrack := TRUE;
END_METHOD

METHOD GetPositionOnCurrentPart : BOOL
VAR_IN_OUT
	position : PositionXYC;
END_VAR
stMoverRef.GetPositionOnCurrentPart(position);
GetPositionOnCurrentPart := TRUE;
END_METHOD

METHOD Halt : BOOL
VAR_INPUT
	slogMessage		: STRING;
END_VAR

VAR_INST
	DynamicConstraint_PathXY 	: DynamicConstraint_PathXY;
	DynamicConstraint_Axis 		: DynamicConstraint_Coordinates;	
	DynamicConstraintStop 		: DynamicConstraint_Container;
	
	stCommand: ST_MoverCommand;
END_VAR
	MEMSET(ADR(stRtHalt), 0, SIZEOF(stRtHalt));

	
	IF 	stHaltDynamics.Mode = E_HaltDynamicsMode.AxisX_AxisY_CoordinatedOnPath THEN
		DynamicConstraint_PathXY.SetValuesVADJ(stHaltDynamics.PathXY.fVelocity, stHaltDynamics.PathXY.fAcceleration, stHaltDynamics.PathXY.fDeceleration, stHaltDynamics.PathXY.fJerk);
	ELSE
		DynamicConstraint_Axis.SetLimit(Coord_Mcs_X, stHaltDynamics.AxisX.fVelocity, stHaltDynamics.AxisX.fAcceleration, stHaltDynamics.AxisX.fDeceleration, stHaltDynamics.AxisX.fJerk);
		DynamicConstraint_Axis.SetLimit(Coord_Mcs_Y, stHaltDynamics.AxisY.fVelocity, stHaltDynamics.AxisY.fAcceleration, stHaltDynamics.AxisY.fDeceleration, stHaltDynamics.AxisY.fJerk);
	END_IF
	DynamicConstraint_Axis.SetLimit(Coord_Mcs_Z,  stHaltDynamics.AxisZ.fVelocity, stHaltDynamics.AxisZ.fAcceleration, stHaltDynamics.AxisZ.fDeceleration, stHaltDynamics.AxisZ.fJerk);
	DynamicConstraint_Axis.SetLimit(Coord_Mcs_A1, stHaltDynamics.AxisA.fVelocity, stHaltDynamics.AxisA.fAcceleration, stHaltDynamics.AxisA.fDeceleration, stHaltDynamics.AxisA.fJerk);
	DynamicConstraint_Axis.SetLimit(Coord_Mcs_B1, stHaltDynamics.AxisB.fVelocity, stHaltDynamics.AxisB.fAcceleration, stHaltDynamics.AxisB.fDeceleration, stHaltDynamics.AxisB.fJerk);
	DynamicConstraint_Axis.SetLimit(Coord_Mcs_C1, stHaltDynamics.AxisC.fVelocity, stHaltDynamics.AxisC.fAcceleration, stHaltDynamics.AxisC.fDeceleration, stHaltDynamics.AxisC.fJerk);
	
	DynamicConstraintStop.Clear();
	DynamicConstraintStop.AddConstraint(DynamicConstraint_PathXY);
	DynamicConstraintStop.AddConstraint(DynamicConstraint_Axis);

	stMoverRef.Halt(haltCmdFB,DynamicConstraintStop); 
	

	
	// Command History
	stCommand.eCommandType 						:= eMoverCommand_eHalt;
	stCommand.sStation							:= slogMessage;
	stCommand.stHaltParameter.fDeceleration_XY  := stHaltDynamics.PathXY.fDeceleration;
	stCommand.stHaltParameter.fJerk_XY			:= stHaltDynamics.PathXY.fJerk;
	stCommand.stHaltParameter.fDeceleration_A	:= stHaltDynamics.AxisA.fDeceleration;
	stCommand.stHaltParameter.fJerk_A			:= stHaltDynamics.AxisA.fJerk;
	stCommand.stHaltParameter.fDeceleration_B	:= stHaltDynamics.AxisB.fDeceleration;
	stCommand.stHaltParameter.fJerk_B			:= stHaltDynamics.AxisB.fJerk;
	stCommand.stHaltParameter.fDeceleration_C	:= stHaltDynamics.AxisC.fDeceleration;
	stCommand.stHaltParameter.fJerk_C			:= stHaltDynamics.AxisC.fJerk;	
	UpdateCommandHistory(stCommand); 
	
	
	Halt := TRUE;
END_METHOD

METHOD JoinTrack : BOOL
VAR_INPUT
	slogMessage		: STRING;
	ipTrack 		: I_TrackStandard;
	fVelo			: LREAL;
	fAcceleration	: LREAL;
	fJerk			: LREAL;
	stOptions		: REFERENCE TO ST_JoinTrackOptions;
END_VAR
	
VAR_INST
	DynamicConstraintPath 	: DynamicConstraint_PathXY;    
END_VAR

VAR
	stCommand 				: ST_MoverCommand;		
	ref 					: POINTER TO MC_PlanarTrack;
END_VAR


VAR_INST
	nState			: INT;
	fbR_TrigExecute : R_TRIG;
	bBusy 			: BOOL;
	bError 			: BOOL;
END_VAR
MEMSET(ADR(stRtJoinTrack), 0, SIZEOF(stRtJoinTrack));
ref := ipTrack.ref;
DynamicConstraintPath.SetValuesVADJ(fvelo,facceleration,facceleration,fjerk);
stMoverRef.JoinTrack(joinTrackCmdFB, ref^, DynamicConstraintPath, stOptions );


// Command History
stCommand.eCommandType 						:= eMoverCommand_eJoinTrack;
stCommand.stJoinTrackParameter.nTargetTrack := ref^.MCTOPLC_STD.TrackOID;
stCommand.stJoinTrackParameter.fVelo		:= fVelo;
stCommand.stJoinTrackParameter.fAcc			:= fAcceleration;
stCommand.stJoinTrackParameter.fJerk		:= fJerk;
stCommand.sStation							:= slogMessage;
UpdateCommandHistory(stCommand);

	
JoinTrack := True;
END_METHOD

METHOD LeaveTrack : BOOL
VAR_INPUT
	slogMessage		: STRING;
	position 		: REFERENCE TO PositionXYC;
	velocity 		: LREAL;
	acceleration	: LREAL;
	deceleration	: LREAL;
	jerk			: LREAL;
	stOptions		: REFERENCE TO ST_LeaveTrackOptions;
END_VAR

VAR_INST
	DynamicConstraintPath : DynamicConstraint_PathXY; 
END_VAR

VAR
	stCommand : ST_MoverCommand;		
END_VAR

VAR_INST
	tempPos : PositionXYC;
END_VAR
MEMSET(ADR(stRtLeaveTrack), 0, SIZEOF(stRtLeaveTrack));

DynamicConstraintPath.SetValuesVADJ(velocity,acceleration,deceleration,jerk);
tempPos.SetValues(position);
stMoverRef.LeaveTrack(leaveTrackCmdFB, position,DynamicConstraintPath, stOptions);




// Command History
stCommand.eCommandType 						:= eMoverCommand_eLeaveTrack;
stCommand.stLeaveTrackParameter.fPositionX  := position.x;
stCommand.stLeaveTrackParameter.fPositionY  := position.y;
stCommand.stLeaveTrackParameter.fPositionC  := position.c;
stCommand.stLeaveTrackParameter.fVelo		:= velocity;
stCommand.stLeaveTrackParameter.fAcc		:= acceleration;
stCommand.stLeaveTrackParameter.fDec		:= deceleration;
stCommand.stLeaveTrackParameter.fJerk		:= jerk;
stCommand.sStation							:= slogMessage;
UpdateCommandHistory(stCommand);


LeaveTrack := TRUE;
END_METHOD

METHOD LeaveTrackInPosition : BOOL
VAR_INPUT
	slogMessage		: STRING;
	bUseOrientation	: BOOL;
END_VAR


VAR_INST
	DynamicConstraintPath : DynamicConstraint_PathXY; 

	velocity 		: LREAL;
	acceleration	: LREAL;
	deceleration	: LREAL;
	jerk			: LREAL;
	currentPos		: MoverVector;

	position 		: PositionXYC;
	stOptions		: ST_LeaveTrackOptions;
	stCommand 		: ST_MoverCommand;		
END_VAR

VAR_INST
	tempPos : PositionXYC;
END_VAR
MEMSET(ADR(LeaveTrackInPosition), 0, SIZEOF(LeaveTrackInPosition));


		velocity := 100.0;
	acceleration := 1000.0;
	deceleration := 1000.0;
			jerk := 10000.0;

	stOptions.useOrientation := bUseOrientation;
 
	
	currentPos := stMoverRef.MCTOPLC.SET.SetPos;
	position.SetValuesXYC(currentPos.x, currentPos.y, currentPos.c);	
		
	
	DynamicConstraintPath.SetValuesVADJ(velocity,acceleration,deceleration,jerk);
	tempPos.SetValues(position);
	stMoverRef.LeaveTrack(leaveTrackInPositionCmdFB, position,DynamicConstraintPath, stOptions);


// Command History
stCommand.eCommandType 								  := eMoverCommand_eLeaveTrackInPosition;
stCommand.stLeaveTrackInPositionParameter.fPositionX  := position.x;
stCommand.stLeaveTrackInPositionParameter.fPositionY  := position.y;
stCommand.stLeaveTrackInPositionParameter.fPositionC  := position.c;
stCommand.sStation									  := slogMessage;
UpdateCommandHistory(stCommand);


LeaveTrackInPosition := TRUE;
END_METHOD

METHOD MoveA : BOOL
VAR_INPUT
	slogMessage		: STRING;
	targetPosition	: LREAL;
	velocity		: LREAL;
	acceleration	: LREAL;
	deceleration	: LREAL;
	jerk			: LREAL;
END_VAR

VAR_INST
	dyn	: DynamicConstraint_Coordinates;  
END_VAR

VAR  
	stMoveToPositionOptions		: ST_MoveToPositionOptions;
	stCommand 					: ST_MoverCommand;
END_VAR
MEMSET(ADR(stRtMoveA), 0, SIZEOF(stRtMoveA));
dyn.SetLimit(Coord_Mcs_A1, velocity, acceleration, deceleration, jerk);
stMoverRef.MoveA(moveACmdFB, targetPosition, dyn);


	
// Command History
stCommand.eCommandType 								:= eMoverCommand_eMoveA;
stCommand.sStation 									:= slogMessage;
stcommand.stMoveOnTrackParameter.fTargetPosition 	:= targetPosition;
stCommand.stMoveOnTrackParameter.fVelo 				:= velocity;
stCommand.stMoveOnTrackParameter.fAcc 				:= acceleration;
stCommand.stMoveOnTrackParameter.fDec 				:= deceleration;
stCommand.stMoveOnTrackParameter.fJerk 				:= jerk;
UpdateCommandHistory(stCommand);



MoveA := TRUE;
END_METHOD

METHOD MoveB : BOOL
VAR_INPUT
	slogMessage		: STRING;
	targetPosition	: LREAL;
	velocity		: LREAL;
	acceleration	: LREAL;
	deceleration	: LREAL;
	jerk			: LREAL;
END_VAR


VAR_INST
	dyn	: DynamicConstraint_Coordinates;  
END_VAR

VAR
	stMoveToPositionOptions		: ST_MoveToPositionOptions;
	stCommand 					: ST_MoverCommand;
END_VAR
MEMSET(ADR(stRtMoveB), 0, SIZEOF(stRtMoveB));
dyn.SetLimit(Coord_Mcs_B1, velocity, acceleration, deceleration, jerk);
stMoverRef.MoveB(moveBCmdFB, targetPosition, dyn);


// Command History
stCommand.eCommandType 								:= eMoverCommand_eMoveB;
stCommand.sStation 									:= slogMessage;
stcommand.stMoveOnTrackParameter.fTargetPosition 	:= targetPosition;
stCommand.stMoveOnTrackParameter.fVelo 				:= velocity;
stCommand.stMoveOnTrackParameter.fAcc 				:= acceleration;
stCommand.stMoveOnTrackParameter.fDec 				:= deceleration;
stCommand.stMoveOnTrackParameter.fJerk 				:= jerk;
UpdateCommandHistory(stCommand);


MoveB := TRUE;
END_METHOD

METHOD MoveC : BOOL
VAR_INPUT
	slogMessage		: STRING;
	targetPosition	: LREAL;
	velocity		: LREAL;
	acceleration	: LREAL;
	deceleration	: LREAL;
	jerk			: LREAL;
	stOptions 		: REFERENCE TO ST_MoveCOptions;
END_VAR


VAR_INST
	dyn	: DynamicConstraint_Coordinates;  
END_VAR

VAR
	stMoveToPositionOptions		: ST_MoveToPositionOptions;
	stCommand 					: ST_MoverCommand;
END_VAR
MEMSET(ADR(stRtMoveC), 0, SIZEOF(stRtMoveC));

//dyn.AddLimit(Coord_Mcs_C1,velocity, acceleration, deceleration, jerk);
dyn.SetLimit(Coord_Mcs_C1,velocity, acceleration, deceleration, jerk);

stMoverRef.MoveC(moveCCmdFB, targetPosition, dyn, stOptions);


// Command History
stCommand.eCommandType 								:= eMoverCommand_eMoveC;
stCommand.sStation 									:= slogMessage;
stcommand.stMoveOnTrackParameter.fTargetPosition 	:= targetPosition;
stCommand.stMoveOnTrackParameter.fVelo 				:= velocity;
stCommand.stMoveOnTrackParameter.fAcc 				:= acceleration;
stCommand.stMoveOnTrackParameter.fDec 				:= deceleration;
stCommand.stMoveOnTrackParameter.fJerk 				:= jerk;
UpdateCommandHistory(stCommand);
	
MoveC := TRUE;
END_METHOD

METHOD MoveOnTrackExt : BOOL
VAR_INPUT
	sLogMessage				: STRING;
	ipTrack					: I_TrackStandard;
	trackPosition       	: LREAL;
	velocity           		: LREAL;
	acceleration        	: LREAL;
	jerk                	: LREAL;
	stMoveOnTrackOptions	: ST_MoveOnTrackOptions;
END_VAR


VAR_INST 
	dyn : DynamicConstraint_PathXY;	 
END_VAR

VAR 
	stCommand 			: ST_MoverCommand; 
	fAbsolutePositon 	: LREAL; // 
	xCommandMissed		: BOOL;
	ref 				: POINTER TO MC_PlanarTrack; 
	//stOptions			: ST_MoveAbsoluteCAOptions; 
END_VAR

VAR_INST
	_ipTrack			: I_TrackStandard;
	_trackPosition      : LREAL;
	_velocity           : LREAL;
	_acceleration       : LREAL;
	_jerk               : LREAL;
	_ref				: POINTER TO MC_PlanarTrack; 
	
	idx					: UDINT;
	nTrackID			: UDINT;
	

END_VAR
MEMSET(ADR(stRtMoveOnTrackExt), 0, SIZEOF(stRtMoveOnTrackExt));

ref := ipTrack.ref;

_ref				:= ref;
_trackPosition      := trackPosition;
_velocity           := velocity;
_acceleration       := acceleration;
_jerk               := jerk;


dyn.SetValuesVADJ(velocity, acceleration, acceleration, jerk); 
stMoverRef.MoveOnTrack(moveOnTrackExtCmdFB, ref^, trackPosition, dyn, stMoveOnTrackOptions);


// Command History
stCommand.eCommandType                               := eMoverCommand_eMoveModOnTrackExt;
stCommand.sStation                                   := sLogMessage;
stCommand.stMoveOnTrackParameterExt.fTargetPosition  := trackPosition ;
stCommand.stMoveOnTrackParameterExt.nTargetTrackOid  := ref^.MCTOPLC_STD.TrackOID;
stCommand.stMoveOnTrackParameterExt.nTargetTrackID   := nTrackID;
stCommand.stMoveOnTrackParameterExt.fAcc 	         := acceleration;
stCommand.stMoveOnTrackParameterExt.fDec 	         := acceleration;
stCommand.stMoveOnTrackParameterExt.fJerk 	         := jerk;
stCommand.stMoveOnTrackParameterExt.fVelo 	         := velocity;
//stCommand.stMoveOnTrackParameter.fGap 	         := gap;
stCommand.stActualParameter 			         	 := UpdateActualMotionParameter();
UpdateCommandHistory(stCommand);


MoveOnTrackExt := TRUE;
END_METHOD

METHOD MoveToPositionExt  : BOOL
VAR_INPUT
	slogMessage					: STRING;
	targetPosition				: REFERENCE TO PositionXYC;
	velocity					: LREAL;
	acceleration				: LREAL;
	deceleration				: LREAL;
	jerk						: LREAL;
	stMoveToPositionOptions		: ST_MoveToPositionOptions;
END_VAR


VAR_INST
	DynamicConstraintPath : DynamicConstraint_PathXY;   
END_VAR

VAR 
	stCommand 					: ST_MoverCommand;	
	stCommandReturnClear		: ST_CommandReturn;
END_VAR
MEMSET(ADR(stRtMoveToPosExt), 0, SIZEOF(stRtMoveToPosExt));
DynamicConstraintPath.SetValuesVADJ(velocity,acceleration,deceleration,jerk);

stMoverRef.MoveToPosition(moveToPosExtCmdFB, targetPosition,  DynamicConstraintPath, stMoveToPositionOptions);


// Command History
stCommand.eCommandType 									:= eMoverCommand_eMoveToPositionExt;
stCommand.sText        									:= slogMessage;
stCommand.stMoveToPositionExt.fTargetPositionX 			:= targetPosition.x;
stCommand.stMoveToPositionExt.fTargetPositionY 			:= targetPosition.y;
stCommand.stMoveToPositionExt.fTargetPositionC 			:= targetPosition.c;
stCommand.stMoveToPositionExt.fVelo						:= DynamicConstraintPath.V;
stCommand.stMoveToPositionExt.fAcc 						:= DynamicConstraintPath.A;
stCommand.stMoveToPositionExt.fDec 						:= DynamicConstraintPath.D;
stCommand.stMoveToPositionExt.fJerk 					:= DynamicConstraintPath.J;
stCommand.stMoveToPositionExt.stMoveToPositionOptions 	:= stMoveToPositionOptions;
UpdateCommandHistory(stCommand);


stRtMoveToPosExt := stCommandReturnClear;


MoveToPositionExt := TRUE;
END_METHOD

{attribute 'hide'}
{attribute 'obsolete' := 'Obsolete: Please use MoveToPositionExt instead'}
METHOD MoveToPositionXYC  : BOOL
VAR_INPUT
	slogMessage		: STRING;
	targetPosition	: REFERENCE TO PositionXYC;
	velocity		: LREAL;
	acceleration	: LREAL;
	deceleration	: LREAL;
	jerk			: LREAL;
END_VAR


VAR_INST
	DynamicConstraintPath : DynamicConstraint_PathXY;   
END_VAR

VAR
	stMoveToPositionOptions		: ST_MoveToPositionOptions;
	stCommand 					: ST_MoverCommand;		
END_VAR
MEMSET(ADR(stRtMoveToPosXYC), 0, SIZEOF(stRtMoveToPosXYC));
DynamicConstraintPath.SetValuesVADJ(velocity,acceleration,deceleration,jerk);




stMoveToPositionOptions.useOrientation := TRUE;
stMoverRef.MoveToPosition(moveToPosXYCCmdFB, targetPosition,  DynamicConstraintPath, stMoveToPositionOptions);



// Command History
stCommand.eCommandType 							:= eMoverCommand_eMoveToPositionXYC;
stCommand.sText        							:= slogMessage;
stCommand.stMoveToPositionXYC.fTargetPositionX 	:= targetPosition.x;
stCommand.stMoveToPositionXYC.fTargetPositionY 	:= targetPosition.y;
stCommand.stMoveToPositionXYC.fTargetPositionC 	:= targetPosition.c;
stCommand.stMoveToPositionXYC.fVelo				:= DynamicConstraintPath.V;
stCommand.stMoveToPositionXYC.fAcc 				:= DynamicConstraintPath.A;
stCommand.stMoveToPositionXYC.fDec 				:= DynamicConstraintPath.D;
stCommand.stMoveToPositionXYC.fJerk 			:= DynamicConstraintPath.J;
UpdateCommandHistory(stCommand);


MoveToPositionXYC := TRUE;
END_METHOD

METHOD MoveZ : BOOL
VAR_INPUT
	slogMessage		: STRING;
	targetPosition	: LREAL;
	velocity		: LREAL;
	acceleration	: LREAL;
	deceleration	: LREAL;
	jerk			: LREAL;
END_VAR

VAR_INST
	dyn	: DynamicConstraint_Coordinates;
END_VAR

VAR
	stMoveToPositionOptions		: ST_MoveToPositionOptions;
	stCommand 					: ST_MoverCommand;
END_VAR
MEMSET(ADR(stRtMoveZ), 0, SIZEOF(stRtMoveZ));

dyn.SetLimit(Coord_Mcs_Z, velocity, acceleration, deceleration, jerk);

stMoverRef.MoveZ(moveZCmdFB, targetPosition, dyn);


// Command History
stCommand.eCommandType 								:= eMoverCommand_eMoveZ;
stCommand.sStation 									:= slogMessage;
stcommand.stMoveOnTrackParameter.fTargetPosition 	:= targetPosition;
stCommand.stMoveOnTrackParameter.fVelo 				:= velocity;
stCommand.stMoveOnTrackParameter.fAcc 				:= acceleration;
stCommand.stMoveOnTrackParameter.fDec 				:= deceleration;
stCommand.stMoveOnTrackParameter.fJerk 				:= jerk;
UpdateCommandHistory(stCommand);


MoveZ := TRUE;
END_METHOD

METHOD RemoveFromGroup : BOOL
VAR_INPUT
END_VAR


VAR
	stCommand : ST_MoverCommand;
END_VAR
MEMSET(ADR(stRtRemoveMover), 0, SIZEOF(stRtRemoveMover));
stMoverRef.RemoveFromGroup(removeMoverCmdFB);

RemoveFromGroup := TRUE;



// Command History
stCommand.eCommandType 	:= eMoverCommand_eRemoveMoverFromGroup;
UpdateCommandHistory(stCommand);
END_METHOD

METHOD Reset : BOOL
VAR_INPUT
	slogMessage 	: STRING;
END_VAR


VAR
	stCommand : ST_MoverCommand;
END_VAR
MEMSET(ADR(stRtReset), 0, SIZEOF(stRtReset));
stMoverRef.Reset(resetCmdFB);

// Command History
stCommand.eCommandType 	:= eMoverCommand_eReset;
stCommand.sText     	:= sLogMessage;
UpdateCommandHistory(stCommand);

Reset := TRUE;
END_METHOD

METHOD SetExternalSetpointValues : BOOL
VAR_INPUT
	position 		: MoverVector;
	velocity 		: MoverVector;
	acceleration 	: MoverVector;
END_VAR
stMoverRef.SetExternalSetpoint(position, velocity, acceleration);

SetExternalSetpointValues := TRUE;
END_METHOD

METHOD SetMoverPosition : BOOL
VAR_INPUT
	slogMessage		: STRING;
	position		: REFERENCE TO PositionXYC;
END_VAR

VAR_INST
	stCommand: ST_MoverCommand;
END_VAR
	MEMSET(ADR(stRtSetMoverPosition), 0, SIZEOF(stRtSetMoverPosition));

	stMoverRef.SetPosition(setMoverPositionCmdFB, position);

	// Command History
	stCommand.eCommandType 				:= eMoverCommand_eSetPosition;
	stCommand.stSetPosition.fPositionX 	:= position.x;
	stCommand.stSetPosition.fPositionY 	:= position.y;
	stCommand.stSetPosition.fPositionC 	:= position.c;
	stCommand.sText 					:= slogMessage;
	
	UpdateCommandHistory(stCommand); 
	
	SetMoverPosition := TRUE;
END_METHOD

METHOD PRIVATE CopyReturnStructure : ST_CommandReturn
VAR_INPUT
	mcInStructur : REFERENCE TO MC_PlanarFeedback;
END_VAR
mcInStructur.Update();
CopyReturnStructure.Active				:= mcInStructur.Active; 
CopyReturnStructure.Busy				:= mcInStructur.Busy;
CopyReturnStructure.Aborted				:= mcInStructur.Aborted;
CopyReturnStructure.Done				:= mcInStructur.Done;
CopyReturnStructure.Error				:= mcInStructur.Error;
CopyReturnStructure.ErrorID 			:= mcInStructur.ErrorId;
CopyReturnStructure.stInfo.nObjectID	:= mcInStructur.objectInfo.Id;
CopyReturnStructure.stInfo.nObjectType	:= mcInStructur.objectInfo.ObjectType;
END_METHOD

METHOD PRIVATE CopyReturnStructureGearInPosOnTrack : ST_CommandReturnGearInPosOnTrack
VAR_INPUT
	mcInStructur : REFERENCE TO MC_PlanarFeedbackGearInPosOnTrack;
END_VAR
mcInStructur.Update();
CopyReturnStructureGearInPosOnTrack.Active				:= mcInStructur.Active; 
CopyReturnStructureGearInPosOnTrack.Busy				:= mcInStructur.Busy;
CopyReturnStructureGearInPosOnTrack.Aborted				:= mcInStructur.Aborted;
//CopyReturnStructureGearInPosOnTrack.Done				:= mcInStructur.Done;
CopyReturnStructureGearInPosOnTrack.Error				:= mcInStructur.Error;
CopyReturnStructureGearInPosOnTrack.ErrorID 			:= mcInStructur.ErrorId;
CopyReturnStructureGearInPosOnTrack.stInfo.nObjectID	:= mcInStructur.objectInfo.Id;
CopyReturnStructureGearInPosOnTrack.stInfo.nObjectType	:= mcInStructur.objectInfo.ObjectType;
CopyReturnStructureGearInPosOnTrack.inSync 				:= mcInStructur.inSync;
END_METHOD

METHOD PRIVATE CopyReturnStructureGearInPosOnTrackMasterMover : ST_CommandReturnGearInPosOnTrackWithMasterMover
VAR_INPUT
	mcInStructur : REFERENCE TO MC_PlanarFeedbackGearInPosOnTrackWithMasterMover;
END_VAR
mcInStructur.Update();
CopyReturnStructureGearInPosOnTrackMasterMover.Active				:= mcInStructur.Active; 
CopyReturnStructureGearInPosOnTrackMasterMover.Busy					:= mcInStructur.Busy;
CopyReturnStructureGearInPosOnTrackMasterMover.Aborted				:= mcInStructur.Aborted;
//CopyReturnStructureGearInPosOnTrackMasterMover.Done				:= mcInStructur.Done;
CopyReturnStructureGearInPosOnTrackMasterMover.Error				:= mcInStructur.Error;
CopyReturnStructureGearInPosOnTrackMasterMover.ErrorID 				:= mcInStructur.ErrorId;
CopyReturnStructureGearInPosOnTrackMasterMover.stInfo.nObjectID		:= mcInStructur.objectInfo.Id;
CopyReturnStructureGearInPosOnTrackMasterMover.stInfo.nObjectType	:= mcInStructur.objectInfo.ObjectType;
CopyReturnStructureGearInPosOnTrackMasterMover.inSync 				:= mcInStructur.inSync;
END_METHOD

METHOD PRIVATE UpdateActualMotionParameter : ST_ActualMotionParameters
VAR_INPUT
END_VAR
UpdateActualMotionParameter.Position			:= stMoverRef.MCTOPLC.SET.SetPos;	
UpdateActualMotionParameter.fSetTrackPosition 	:= stMoverRef.MCTOPLC.SETONTRACK.SetPos;	
UpdateActualMotionParameter.nTrackOid 		  	:= stMoverRef.MCTOPLC.SETONTRACK.TrackOID;	
UpdateActualMotionParameter.sTrackName 		  	:= '';		
UpdateActualMotionParameter.fSetVelo			:= stMoverRef.MCTOPLC.SETONTRACK.SetVelo;
UpdateActualMotionParameter.fSetAcc				:= stMoverRef.MCTOPLC.SETONTRACK.SetAcc;
END_METHOD

PROPERTY P_AtRotationPoint : BOOL
GET
P_AtRotationPoint := bAtRotationPoint;
END_GET
END_PROPERTY

PROPERTY P_ClosestQuaterAngle : LREAL
GET
P_ClosestQuaterAngle := fClosestQuaterAngle;
END_GET
END_PROPERTY

PROPERTY P_CRotationRestrictions : BOOL
GET
P_CRotationRestrictions := bCRotationRestrictions;
END_GET
END_PROPERTY

PROPERTY P_CustomTrackIdTable : ARRAY [1..Params_XPlanar.maxTrackCount] OF ST_CutomTrackID;
SET
CustomTrackIdTable := P_CustomTrackIdTable;
END_SET
END_PROPERTY

PROPERTY P_HaltDynamics : ST_HaltDynamics
GET
P_HaltDynamics := stHaltDynamics;
END_GET
SET
stHaltDynamics := P_HaltDynamics;
END_SET
END_PROPERTY

PROPERTY P_IsMovingXY : BOOL
GET
P_isMovingXY := bIsMovingXY;
END_GET
END_PROPERTY

PROPERTY P_IsPresent : BOOL
GET
IF stMoverRef.MCTOPLC.ACT.PhysicalAreaID > 0 THEN
	P_IsPresent := TRUE;
ELSE
	p_IsPresent := FALSE;
END_IF
END_GET
END_PROPERTY

PROPERTY P_IsQueuing : BOOL
GET

P_IsQueuing := bIsQueuing;
END_GET
END_PROPERTY

PROPERTY P_IsSetpointGeneratorActive : BOOL
GET
P_IsSetpointGeneratorActive := bIsSetpointGeneratorActive;
END_GET
END_PROPERTY

PROPERTY P_LastKnownTrackOID : OTCID
GET
P_LastKnownTrackOID := nLastKnownTrackOID;
END_GET
END_PROPERTY

PROPERTY P_RotationAngleModulo : LREAL
GET

P_RotationAngleModulo := fCurrentAngleC_Modulo;
END_GET
END_PROPERTY

PROPERTY P_SavedMoveOnTrackParameter : REFERENCE TO ST_MoveOnTrackParameters
GET
P_SavedMoveOnTrackParameter REF= stMoveOnTrackParameter;
END_GET
END_PROPERTY


PROPERTY P_ZeroVelocityThreshold : LREAL
GET
P_ZeroVelocityThreshold := fZeroVelocityThreshold;
END_GET
SET
fZeroVelocityThreshold := ABS(P_ZeroVelocityThreshold);
END_SET
END_PROPERTY

PROPERTY P_AddToGroup : REFERENCE to ST_CommandReturn
GET
P_AddToGroup ReF= stRtAddMover;
END_GET
END_PROPERTY

PROPERTY P_AdoptTrackOrientation : REFERENCE TO ST_CommandReturn
GET
P_AdoptTrackOrientation REF= stRtAdoptTrackOri;
END_GET
END_PROPERTY

PROPERTY P_Disable : REFERENCE to ST_CommandReturn
GET
P_Disable ReF= stRtDisable;
END_GET
END_PROPERTY

PROPERTY P_DisableExternalSetpointGeneration : REFERENCE to ST_CommandReturn
GET
P_DisableExternalSetpointGeneration ReF= stRtDisableSetPos;
END_GET
END_PROPERTY

PROPERTY P_Enable : REFERENCE to ST_CommandReturn
GET
P_Enable ReF= stRtEnable;
END_GET
END_PROPERTY

PROPERTY P_EnableExternalSetpointGeneration : REFERENCE to ST_CommandReturn
GET
P_EnableExternalSetpointGeneration ReF= stRtEnableSetPos;
END_GET
END_PROPERTY

PROPERTY P_GearInPosOnTrack : REFERENCE TO ST_CommandReturnGearInPosOnTrack
GET
P_GearInPosOnTrack REF= stRtGearInPosOnTrack;
END_GET
END_PROPERTY

PROPERTY P_GearInPosOnTrackMasterMover : REFERENCE TO ST_CommandReturnGearInPosOnTrackWithMasterMover
GET
P_GearInPosOnTrackMasterMover REF= stRtGearInPosOnTrackMasterMover;
END_GET
END_PROPERTY

PROPERTY P_Halt : REFERENCE to ST_CommandReturn
GET
P_Halt ReF= stRtHalt;
END_GET
END_PROPERTY

PROPERTY P_JoinTrack : REFERENCE to ST_CommandReturn
GET
P_JoinTrack ReF= stRtJoinTrack;
END_GET
END_PROPERTY

PROPERTY P_LeaveTrack : REFERENCE to ST_CommandReturn
GET
P_LeaveTrack ReF= stRtLeaveTrack;
END_GET
END_PROPERTY

PROPERTY P_LeaveTrackInPosition : REFERENCE to ST_CommandReturn
GET
P_LeaveTrackInPosition ReF= stRtLeaveTrackInPosition;
END_GET
END_PROPERTY

PROPERTY P_MoveA : REFERENCE to ST_CommandReturn
GET
P_MoveA ReF= stRtMoveA;
END_GET
END_PROPERTY

PROPERTY P_MoveB : REFERENCE to ST_CommandReturn
GET
P_MoveB ReF= stRtMoveB;
END_GET
END_PROPERTY

PROPERTY P_MoveC : REFERENCE TO ST_CommandReturn
GET
P_MoveC ReF= stRtMoveC;
END_GET
END_PROPERTY

PROPERTY P_MoveOnTrack : REFERENCE to ST_CommandReturn
GET
P_MoveOnTrack ReF= stRtMoveOnTrack;
END_GET
END_PROPERTY

PROPERTY P_MoveOnTrackExt : REFERENCE to ST_CommandReturn
GET
P_MoveOnTrackExt ReF= stRtMoveOnTrackExt;
END_GET
END_PROPERTY

{attribute 'obsolete' := 'Obsolete: Please use P_MoveToPositionExt instead'}
PROPERTY P_MoveToPosition : REFERENCE to ST_CommandReturn
GET
P_MoveToPosition ReF= stRtMoveToPos;
END_GET
END_PROPERTY


PROPERTY P_MoveToPositionExt : REFERENCE to ST_CommandReturn
GET
P_MoveToPositionExt ReF= stRtMoveToPosExt;
END_GET
END_PROPERTY

{attribute 'hide'}
{attribute 'obsolete' := 'Obsolete: Please use P_MoveToPositionExt instead'}
PROPERTY P_MoveToPositionXYC : REFERENCE to ST_CommandReturn
GET
P_MoveToPositionXYC ReF= stRtMoveToPosXYC;
END_GET
END_PROPERTY

PROPERTY P_MoveZ : REFERENCE to ST_CommandReturn
GET
P_MoveZ ReF= stRtMoveZ;
END_GET
END_PROPERTY

PROPERTY P_RemoveFromGroup : REFERENCE TO ST_CommandReturn
GET
P_RemoveFromGroup REF= stRtRemoveMover;
END_GET
END_PROPERTY

PROPERTY P_Reset : REFERENCE to ST_CommandReturn
GET
P_Reset ReF= stRtReset;
END_GET
END_PROPERTY


PROPERTY P_SetMoverPosition : REFERENCE to ST_CommandReturn
GET
P_SetMoverPosition ReF= stRtSetMoverPosition;
END_GET
END_PROPERTY

PROPERTY P_ActPosition : REFERENCE TO MoverVector
GET
ActPos :=  stMoverRef.MCTOPLC.ACT.ActPos;

P_ActPosition REF= ActPos;
END_GET
END_PROPERTY

PROPERTY P_ActVelocity : REFERENCE TO MoverVector
GET
ActVelo :=  stMoverRef.MCTOPLC.ACT.ActVelo;

P_ActVelocity REF= ActVelo;
END_GET
END_PROPERTY

PROPERTY P_Busy : BOOL
GET
P_Busy := stMoverRef.MCTOPLC.STD.Busy.busyMover;
END_GET
END_PROPERTY

PROPERTY P_CommandMode : MC_PLANAR_MOVER_COMMAND_MODE;
GET
P_CommandMode  := stMoverRef.MCTOPLC.STD.CommandMode;
END_GET
END_PROPERTY

PROPERTY P_Error : Bool
GET
P_Error := stMoverRef.Error;
END_GET
END_PROPERTY

PROPERTY P_ErrorCode : DINT
GET
P_ErrorCode := stMoverRef.MCTOPLC.STD.ErrorCode;
END_GET
END_PROPERTY

PROPERTY P_ErrorID : UDINT
GET
P_ErrorID := stMoverRef.ErrorId;
END_GET
END_PROPERTY

PROPERTY P_Id : UINT
GET
P_Id  := nId;
END_GET
SET
nId := P_Id;
END_SET
END_PROPERTY

PROPERTY P_InGroup : BOOL
GET
P_InGroup := bInGroup;
END_GET
END_PROPERTY

PROPERTY P_MoverOid : OTCID
GET
P_MoverOid := stMoverRef.MCTOPLC.STD.MoverOID;
END_GET
END_PROPERTY

{attribute 'hide'}
PROPERTY P_MoverRef : POINTER TO MC_PlanarMover
GET
P_MoverRef := ADR(stMoverRef);
END_GET
END_PROPERTY

PROPERTY P_PhysicalAreaID : UDINT
GET
P_PhysicalAreaID := stMoverRef.MCTOPLC.ACT.PhysicalAreaID;
END_GET
END_PROPERTY

PROPERTY P_SetAcceleration : REFERENCE TO MoverVector
GET


SetAcc :=  stMoverRef.MCTOPLC.SET.SetAcc;
P_SetAcceleration REF= SetAcc;
END_GET
END_PROPERTY

PROPERTY P_SetOnTrack : Reference To CDT_MCTOPLC_PLANAR_MOVER_TRACK
GET


SetOnTrack :=  stMoverRef.MCTOPLC.SETONTRACK;

P_SetOnTrack REF= SetOnTrack;
END_GET
END_PROPERTY

PROPERTY P_SetPosition : Reference To MoverVector
GET
SetPos :=  stMoverRef.MCTOPLC.SET.SetPos;

P_SetPosition REF= SetPos;
END_GET
END_PROPERTY

PROPERTY P_SetVelocity : REFERENCE TO MoverVector
GET
SetVelo :=  stMoverRef.MCTOPLC.SET.SetVelo;

P_SetVelocity REF= SetVelo;
END_GET
END_PROPERTY

PROPERTY P_State : MC_PLANAR_STATE
GET
P_State := stMoverRef.MCTOPLC.STD.State;
END_GET
END_PROPERTY

PROPERTY P_TrackId : UDINT
GET
P_TrackId  := stMoverRef.MCTOPLC.SETONTRACK.TrackOID;
END_GET
END_PROPERTY

METHOD Cycle : BOOL
VAR_INPUT
END_VAR
VAR_INST
	rTrigAddToGroup 		: R_Trig;
	rTrigRemoveFromGroup 	: R_Trig;
	
	fAngleDivisor				: LREAL;
	fCheckAngle					: LREAL;
	fClosestQuaterAngleModulo	: LREAL;
	
	
	CurrentPosition				: MoverVector;
	fCurrentPositionX			: LREAL;
	fCurrentPositionX_Temp		: LREAL;
	fCurrentPositionX_Deviation : LREAL;
	fDividerX					: LREAL;
	bPositionXLimitExceeded		: BOOL;
	
	fCurrentPositionY			: LREAL;
	fCurrentPositionY_Temp		: LREAL;
	fCurrentPositionY_Deviation	: LREAL;
	fDividerY					: LREAL;
	bPositionYLimitExceeded		: BOOL;
	
	

END_VAR


	// Cycle 
	nCycleCounter := nCycleCounter +1;
	stMoverRef.Update();


	// Checking if the mover is in the group
	bInGroup := stMoverRef.MCTOPLC.STD.GroupOID <> 0;
	

	// Check is moving
	CurrentVelocity := stMoverRef.MCTOPLC.SET.SetVelo;	
	IF  ABS(CurrentVelocity.x) > fZeroVelocityThreshold 
	OR  ABS(CurrentVelocity.y) > fZeroVelocityThreshold
	THEN
		bIsMovingXY := TRUE;
	ELSE
		bIsMovingXY := FALSE;
	END_IF	

	
	// Check if the mover is queuing 
	//IF moveOnTrackCmdFB.Busy OR moveOnTrackExtCmdFB.Busy
	IF moveOnTrackCmdFB.Active OR moveOnTrackExtCmdFB.Active
	AND NOT bIsMovingXY
	THEN
		bIsQueuing := TRUE;
	ELSE
		bIsQueuing := FALSE;
	END_IF


	IF stMoverRef.MCTOPLC.SETONTRACK.TrackOID > 0 THEN
		nLastKnownTrackOID := stMoverRef.MCTOPLC.SETONTRACK.TrackOID;
	END_IF
	
	
	
	// Calculating the modulo mover angle c-axis
	      CurrentPosition := stMoverRef.MCTOPLC.ACT.ActPos;
	       fCurrentAngleC := CurrentPosition.c;
			fAngleDivisor := LTRUNC(fCurrentAngleC/360.0);
	fCurrentAngleC_Modulo := fCurrentAngleC - fAngleDivisor * 360.0;

	
	
	// Check for C-Rotation-Restrictions
	bCRotationRestrictions := FALSE;
	fCheckAngle := ABS(fCurrentAngleC_Modulo);
	IF  fCheckAngle > 10.0 	AND fCheckAngle < 80.0
	OR  fCheckAngle > 100.0 AND fCheckAngle < 170.0 
	OR  fCheckAngle > 190.0 AND fCheckAngle < 260.0 
	OR  fCheckAngle > 280.0 AND fCheckAngle < 350.0 
	THEN		
		bCRotationRestrictions := TRUE;
	END_IF


	// Determine closest index angle
	IF fCheckAngle >= 0.0 AND fCheckAngle <= 45.0 THEN
		fClosestQuaterAngleModulo := 0.0;
	ELSIF fCheckAngle > 45.0 AND fCheckAngle <= 90.0 THEN
		fClosestQuaterAngleModulo := 90.0;
	ELSIF fCheckAngle > 90.0 AND fCheckAngle <= 135.0 THEN
		fClosestQuaterAngleModulo := 90.0;
	ELSIF fCheckAngle > 135.0 AND fCheckAngle <= 180.0 THEN
		fClosestQuaterAngleModulo := 180.0;
	ELSIF fCheckAngle > 180.0 AND fCheckAngle <= 225.0 THEN
		fClosestQuaterAngleModulo := 180.0;
	ELSIF fCheckAngle > 225.0 AND fCheckAngle <= 270.0 THEN
		fClosestQuaterAngleModulo := 270.0;
	ELSIF fCheckAngle > 270.0 AND fCheckAngle <= 315.0 THEN
		fClosestQuaterAngleModulo := 270.0;
	ELSIF fCheckAngle > 315.0 AND fCheckAngle <= 360.0 THEN
		fClosestQuaterAngleModulo := 360.0;	
	END_IF	
	IF fCurrentAngleC_Modulo < 0.0 THEN
		fClosestQuaterAngleModulo := -fClosestQuaterAngleModulo;
	END_IF
	fClosestQuaterAngle := fClosestQuaterAngleModulo + fAngleDivisor * 360.0;
	
	

	

	
	// Check if the mover is positioned at a rotation point
	  CurrentPosition := stMoverRef.MCTOPLC.ACT.ActPos;
	fCurrentPositionX := ABS(CurrentPosition.x);
	fCurrentPositionY := ABS(CurrentPosition.y);
	   fCurrentAngleC := ABS(CurrentPosition.c);

	   
	//IF bCRotationRestrictions THEN   
	IF TRUE THEN
		// Position X-Limit
		IF fCurrentPositionX < 120.0
		OR fCurrentPositionX > 120.0
		THEN
			fDividerX := LTRUNC(fCurrentPositionX/120.0);
		ELSE
			fDividerX := 0;
		END_IF
		fCurrentPositionX_Temp := fCurrentPositionX - fDividerX * 120.0;
	
		IF fCurrentPositionX_Temp > 60.0 THEN
			fCurrentPositionX_Deviation := fCurrentPositionX_Temp - 120;
		ELSIF fCurrentPositionX_Temp < -60.0 THEN
			fCurrentPositionX_Deviation := fCurrentPositionX_Temp + 120;
		ELSE
			fCurrentPositionX_Deviation := fCurrentPositionX_Temp;
		END_IF
	
		IF ABS(fCurrentPositionX_Deviation) > 1.0 THEN
			bPositionXLimitExceeded := TRUE;
		ELSE
			bPositionXLimitExceeded := FALSE;
		END_IF
		
	
		// Position Y-Limit
		IF fCurrentPositionY < 120.0
		OR fCurrentPositionY > 120.0
		THEN
			fDividerY := LTRUNC(fCurrentPositionY/120.0);
		ELSE
			fDividerY := 0;
		END_IF
		fCurrentPositionY_Temp := fCurrentPositionY - fDividerY * 120.0;
	
		IF fCurrentPositionY_Temp > 60.0 THEN
			fCurrentPositionY_Deviation := fCurrentPositionY_Temp - 120;
		ELSIF fCurrentPositionY_Temp < -60.0 THEN
			fCurrentPositionY_Deviation := fCurrentPositionY_Temp + 120;
		ELSE
			fCurrentPositionY_Deviation := fCurrentPositionY_Temp;
		END_IF
	
		IF ABS(fCurrentPositionY_Deviation) > 1.0 THEN
			bPositionYLimitExceeded := TRUE;
		ELSE
			bPositionYLimitExceeded := FALSE;
		END_IF		
		bAtRotationPoint := NOT(bPositionXLimitExceeded OR bPositionYLimitExceeded);
	
	ELSE
		IF bPositionXLimitExceeded THEN bPositionXLimitExceeded := FALSE; END_IF
		IF bPositionYLimitExceeded THEN bPositionYLimitExceeded := FALSE; END_IF
		IF bAtRotationPoint THEN bAtRotationPoint := FALSE; END_IF
	END_IF
		
	

	
	// Command-Feedback
	stRtAdoptTrackOri 				:= CopyReturnStructure(adoptTrackOriCmdFb);
	stRtEnable 		  				:= CopyReturnStructure(enableCmdFb);
	stRtDisable 	  				:= CopyReturnStructure(disableCmdFb);
	stRtJoinTrack 	  				:= CopyReturnStructure(joinTrackCmdFb);
	stRtLeaveTrack 	  				:= CopyReturnStructure(leaveTrackCmdFb);
	stRtLeaveTrackInPosition		:= CopyReturnStructure(leaveTrackInPositionCmdFb);
	stRtMoveOnTrack   				:= CopyReturnStructure(moveOnTrackCmdFb);	
	stRtMoveOnTrackExt   			:= CopyReturnStructure(moveOnTrackExtCmdFb);	
	stRtMoveToPos 	  				:= CopyReturnStructure(moveToPosCmdFb);
	stRtMoveToPosXYC 	  			:= CopyReturnStructure(moveToPosXYCCmdFb);
	stRtMoveToPosExt 	  			:= CopyReturnStructure(moveToPosExtCmdFb);
	stRtHalt 		  				:= CopyReturnStructure(haltCmdFb);
	stRtAddMover 	  				:= CopyReturnStructure(addMoverCmdFb); 	
	stRtRemoveMover   				:= CopyReturnStructure(removeMoverCmdFb);
	stRtReset 		  				:= CopyReturnStructure(resetCmdFb);
	stRtMoveZ		  				:= CopyReturnStructure(moveZCmdFb);
	stRtMoveA		  				:= CopyReturnStructure(moveACmdFb);
	stRtMoveB		  				:= CopyReturnStructure(moveBCmdFb);
	stRtMoveC		  				:= CopyReturnStructure(moveCCmdFb);
	stRtEnableSetPos  				:= CopyReturnStructure(enableExtSetPosCmdFB);
	stRtDisableSetPos 				:= CopyReturnStructure(disableExtSetPosCmdFB);
	stRtGearInPosOnTrack 			:= CopyReturnStructureGearInPosOnTrack(gearInPosOnTrackCmdFB);
	stRtGearInPosOnTrackMasterMover := CopyReturnStructureGearInPosOnTrackMasterMover(gearInPosOnTrackMasterMoverCmdFB);
	stRtSetMoverPosition 	  			:= CopyReturnStructure(setMoverPositionCmdFB);

	

	
	IF NOT bInitHaltDynamicsDone THEN
		bInitHaltDynamicsDone := TRUE;	
		
		stHaltDynamics.Mode := E_HaltDynamicsMode.AxisX_AxisY_CoordinatedOnPath;
	
		IF stHaltDynamics.PathXY.fVelocity 		= 0.0 THEN stHaltDynamics.PathXY.fVelocity 		:= 1000.0; 								END_IF
		IF stHaltDynamics.PathXY.fDeceleration 	= 0.0 THEN stHaltDynamics.PathXY.fDeceleration 	:= 10000.0; 							END_IF
		IF stHaltDynamics.PathXY.fAcceleration 	= 0.0 THEN stHaltDynamics.PathXY.fAcceleration 	:= stHaltDynamics.PathXY.fDeceleration; END_IF	
		IF stHaltDynamics.PathXY.fJerk 			= 0.0 THEN stHaltDynamics.PathXY.fJerk 			:= 10000.0; 							END_IF
	
		IF stHaltDynamics.AxisX.fVelocity 		= 0.0 THEN stHaltDynamics.AxisX.fVelocity 		:= 1000.0;								END_IF
		IF stHaltDynamics.AxisX.fDeceleration 	= 0.0 THEN stHaltDynamics.AxisX.fDeceleration 	:= 10000.0; 							END_IF
		IF stHaltDynamics.AxisX.fAcceleration 	= 0.0 THEN stHaltDynamics.AxisX.fAcceleration 	:= stHaltDynamics.PathXY.fDeceleration; END_IF	
		IF stHaltDynamics.AxisX.fJerk			= 0.0 THEN stHaltDynamics.AxisX.fJerk 			:= 10000.0; 							END_IF
	
		IF stHaltDynamics.AxisY.fVelocity		= 0.0 THEN stHaltDynamics.AxisY.fVelocity 		:= 1000.0;								END_IF
		IF stHaltDynamics.AxisY.fDeceleration 	= 0.0 THEN stHaltDynamics.AxisY.fDeceleration 	:= 10000.0; 							END_IF
		IF stHaltDynamics.AxisY.fAcceleration 	= 0.0 THEN stHaltDynamics.AxisY.fAcceleration 	:= stHaltDynamics.PathXY.fDeceleration; END_IF	
		IF stHaltDynamics.AxisY.fJerk 			= 0.0 THEN stHaltDynamics.AxisY.fJerk 			:= 10000.0; 							END_IF
			
		IF stHaltDynamics.AxisZ.fVelocity 		= 0.0 THEN stHaltDynamics.AxisZ.fVelocity 		:= 10.0;							 	END_IF
		IF stHaltDynamics.AxisZ.fDeceleration 	= 0.0 THEN stHaltDynamics.AxisZ.fDeceleration 	:= 100.0;								END_IF
		IF stHaltDynamics.AxisZ.fAcceleration 	= 0.0 THEN stHaltDynamics.Axisz.fAcceleration 	:= stHaltDynamics.PathXY.fDeceleration; END_IF	
		IF stHaltDynamics.AxisZ.fJerk 			= 0.0 THEN stHaltDynamics.AxisZ.fJerk 			:= 100.0; 								END_IF	
		
		IF stHaltDynamics.AxisA.fVelocity 		= 0.0 THEN	stHaltDynamics.AxisA.fVelocity 		:= 1.0;									END_IF
		IF stHaltDynamics.AxisA.fDeceleration 	= 0.0 THEN	stHaltDynamics.AxisA.fDeceleration 	:= 100.0;								END_IF
		IF stHaltDynamics.AxisA.fAcceleration 	= 0.0 THEN	stHaltDynamics.AxisA.fAcceleration 	:= stHaltDynamics.AxisA.fDeceleration;	END_IF		
		IF stHaltDynamics.AxisA.fJerk 			= 0.0 THEN	stHaltDynamics.AxisA.fJerk 			:= 100.0;								END_IF		
		
		IF stHaltDynamics.AxisB.fVelocity 		= 0.0 THEN	stHaltDynamics.AxisB.fVelocity 		:= 1.0;									END_IF
		IF stHaltDynamics.AxisB.fDeceleration	= 0.0 THEN	stHaltDynamics.AxisB.fDeceleration 	:= 100.0;								END_IF
		IF stHaltDynamics.AxisB.fAcceleration 	= 0.0 THEN	stHaltDynamics.AxisB.fAcceleration 	:= stHaltDynamics.AxisB.fDeceleration;	END_IF		
		IF stHaltDynamics.AxisB.fJerk 			= 0.0 THEN	stHaltDynamics.AxisB.fJerk 			:= 100.0;								END_IF			
			
		IF stHaltDynamics.AxisC.fVelocity 		= 0.0 THEN	stHaltDynamics.AxisC.fVelocity 		:= 360.0;								END_IF
		IF stHaltDynamics.AxisC.fDeceleration 	= 0.0 THEN	stHaltDynamics.AxisC.fDeceleration 	:= 3600.0;								END_IF
		IF stHaltDynamics.AxisC.fAcceleration 	= 0.0 THEN	stHaltDynamics.AxisC.fAcceleration 	:= stHaltDynamics.AxisC.fDeceleration;	END_IF		
		IF stHaltDynamics.AxisC.fJerk 			= 0.0 THEN	stHaltDynamics.AxisC.fJerk 			:= 3600.0;								END_IF		
	
	END_IF
END_METHOD

END_FUNCTION_BLOCK

// XPlanarStandardFunctions/MoverQueue/FB_MoverQueue
FUNCTION_BLOCK FB_MoverQueue IMPLEMENTS I_MoverQueue
VAR
	_count	: UDINT;															// Mover currently in queue
	_items	: ARRAY[1..Params_XPlanar.maxNumMover] OF I_XPlanarMoverStandard;	// Mover queue
END_VAR

METHOD Clear
MEMSET(destAddr:= ADR(_items), fillByte:= 0, n:= SIZEOF(_items));

_count := 0;
END_METHOD

METHOD Dequeue : I_XPlanarMoverStandard
VAR_INST
	mover	: I_XPlanarMoverStandard;
	i		: UDINT;
END_VAR
mover := 0;

IF _count > 0 THEN
	// Remove first of the queue and shift remaining in queue
	mover := _items[1];
	_count := _count - 1;

	IF _count > 0 THEN
		FOR i := 1 TO _count DO
			_items[i] := _items[i + 1];
		END_FOR
	END_IF

	// Clear last pos
	_items[_count + 1] := 0;
END_IF

Dequeue := mover;
END_METHOD

METHOD Enqueue : BOOL;
VAR_INPUT
	mover	: I_XPlanarMoverStandard;	// Mover to be added at the end of the queue
END_VAR
IF mover = 0 THEN
	// Invalid Mover itf
	Enqueue := FALSE;
ELSE
	IF _count >= Params_XPlanar.maxNumMover THEN
		// Queue already full
		Enqueue := FALSE;
	ELSE
		// Add Mover as last in list
		_items[_count + 1] := mover;
		_count := _count + 1;
		Enqueue := TRUE;
	END_IF
END_IF
END_METHOD

PROPERTY Count : UDINT
GET
Count := _count;
END_GET
END_PROPERTY

METHOD Item : I_XPlanarMoverStandard
VAR_INPUT
	rank	: UDINT;	// Mover rank (ordinal pos. in queue)
END_VAR
IF rank > _count OR rank < 1 THEN
	Item := 0;
ELSE
	Item := _items[rank];
END_IF
END_METHOD

END_FUNCTION_BLOCK

// XPlanarStandardFunctions/MoverQueue/I_MoverQueue
INTERFACE I_MoverQueue

METHOD Clear
END_METHOD

METHOD Dequeue : I_XPlanarMoverStandard
END_METHOD

METHOD Enqueue : BOOL
VAR_INPUT
	mover	: I_XPlanarMoverStandard;	// Mover to be added at the end of the queue
END_VAR
END_METHOD

PROPERTY Count : UDINT
GET
END_GET
END_PROPERTY

METHOD Item : I_XPlanarMoverStandard
VAR_INPUT
	rank	: UDINT;	// Mover rank (ordinal pos. in queue)
END_VAR
END_METHOD

END_INTERFACE

// XPlanarStandardFunctions/Station/FB_List
FUNCTION_BLOCK FB_List IMPLEMENTS I_List
VAR
	nTrackCount			: UDINT;
	nTrackOIDs			: ARRAY [1..maxTrackCount] OF UDINT;
	TrackList			: ARRAY [1..maxTrackCount] OF I_TrackStandard;
	
	nMoverCount			: UDINT;
	MoversList			: ARRAY [1..maxNumMover] OF ST_MoverInList;
	
	MoversListITF 		: ARRAY[1..maxNumMover] OF I_XPlanarMoverStandard; 
	NoMover				: I_XPlanarMoverStandard;
	
	sStatusMessage		: STRING;
		  nResult		: DINT;
		  

	{attribute 'hide'}
	nSortingMode		: INT;
	nSortingDirection	: eSortingDirection;
	
	fLengthFirstTrack	: LREAL;	
	fSortingOrigin		: LREAL;
	bTrackSplit			: BOOL;

	
	TrackBuiltInfo		: ST_TrackBuiltInfo;

	sHistoryAddMover	: ARRAY[0..10] OF STRING;
END_VAR

{attribute 'hide'}
{attribute 'obsolete' := 'Obsolete: Please use P_SortingDirection instead'}
PROPERTY P_eSortingMode : eSortingMode
GET

IF nSortingDirection = 0 THEN
	P_eSortingMode := eSortingMode.ascending;
ELSE
	P_eSortingMode := eSortingMode.descending;
END_IF
END_GET
SET


IF P_eSortingMode = eSortingMode.ascending THEN
	nSortingDirection := eSortingDirection.ascending;
ELSE
	nSortingDirection := eSortingDirection.descending;
END_IF
END_SET
END_PROPERTY

{attribute 'hide'}
{attribute 'obsolete' := 'Obsolete: Please use P_SortingOrigin instead'}
PROPERTY P_fSortingOrigin : LREAL
GET
P_fSortingOrigin := fSortingOrigin;
END_GET
SET

fSortingOrigin := P_fSortingOrigin;
END_SET
END_PROPERTY

{attribute 'hide'}
{attribute 'obsolete' := 'Obsolete: Please use P_NumberInList instead'}
PROPERTY P_nNumberInList : UDINT
GET
   P_nNumberInList := nMoverCount;
END_GET
END_PROPERTY

{attribute 'hide'}
{attribute 'obsolete' := 'Obsolete: Please use P_Result instead'}
PROPERTY P_nResult : DINT
GET

	P_nResult := nResult;
END_GET
END_PROPERTY

{attribute 'hide'}
{attribute 'obsolete' := 'Obsolete: Please use P_SortingDirection instead'}
PROPERTY P_nSortingMode : INT
GET
P_nSortingMode := nSortingMode;
END_GET
SET
nSortingMode := P_nSortingMode;



// Unfortunately there was a mixup in the older version, that's why we switch the order here for compatibility with older projects.
IF nSortingMode = eSortingMode.ascending THEN
	nSortingDirection := eSortingDirection.descending;
ELSE
	nSortingDirection := eSortingDirection.ascending;
END_IF
END_SET
END_PROPERTY

{attribute 'hide'}
{attribute 'obsolete' := 'Obsolete: Please use P_Message instead'}

PROPERTY P_sMessage : STRING
GET
P_sMessage := sStatusMessage;
END_GET
END_PROPERTY

{attribute 'hide'}
PROPERTY P_SortingMode : eSortingMode
GET


P_SortingMode := nSortingMode;
END_GET
SET

nSortingMode := P_SortingMode;

// Unfortunately there was a mixup in the older version, that's why we switch the order here for compatibility with older projects.
IF nSortingMode = eSortingMode.ascending THEN
	nSortingDirection := eSortingDirection.descending;
ELSE
	nSortingDirection := eSortingDirection.ascending;
END_IF
END_SET
END_PROPERTY

METHOD AddMover : DINT
VAR_INPUT
	ipMover		: I_XPlanarMoverStandard;
END_VAR


VAR_INST
	nMoverIndex	 	: UDINT;
	nMoverPosition 	: LREAL;
	nMoverTrackOID 	: UDINT;

	idx				: UDINT;
	nState	    	: INT;
	bDoubleEntry	: BOOL;
	
	bNewMoverId		: BOOL;
	nMoverItfCount	: UDINT;
	
	nCycleTest	: UINT;
	
	sText		: STRING;
	
END_VAR


	nCycleTest := nCycleTest +1;


	       nResult := 0;
	sStatusMessage := '';
		
	IF ipMover <> 0 THEN
				
		nMoverIndex    := ipMover.P_Id;
		nMoverPosition := ipMover.P_SetOnTrack.SetPos;
		nMoverTrackOID := ipMover.P_SetOnTrack.TrackOID;	
		

		// Check incoming MoverIndex
		IF nResult = 0 THEN
			IF nMoverIndex = 0 THEN
				nResult := -11;
			END_IF
		END_IF
	
		// Check mover Track OID	
		IF nResult = 0 THEN
			IF nMoverTrackOID = 0 THEN
				nResult := -12;
			END_IF
		END_IF
		
		// Check for space
		IF nResult = 0 THEN
			IF nMoverCount >= maxNumMover THEN
				nResult := -13;
			END_IF
		END_IF
			
		// Check for double entry	
		IF nResult = 0 THEN
			bDoubleEntry := FALSE;
			FOR idx:=1 TO nMoverCount DO
				IF MoversList[idx].nMoverIndex = nMoverIndex THEN
					bDoubleEntry := TRUE;
				END_IF
			END_FOR	
			IF bDoubleEntry THEN
				nResult := -14;		
			END_IF
		END_IF
	
	ELSE
		// Invalid input parameter
		nResult := -15;	
	END_IF	
		

	
	// Adding Mover		
	IF nResult >= 0 THEN	
		nMoverCount := nMoverCount +1;
		
		bNewMoverId := TRUE;
		nMoverItfCount := 0;
		FOR idx:=1 TO maxNumMover DO 
			IF MoversListITF[idx] <> 0 THEN
				nMoverItfCount := nMoverItfCount +1;
				IF MoversListITF[idx].P_Id = nMoverIndex THEN
					bNewMoverId := FALSE;	
				END_IF
			END_IF
		END_FOR	
		IF bNewMoverId THEN
			IF (nMoverItfCount+1) <= maxNumMover THEN
				MoversListITF[nMoverItfCount+1] := ipMover;
			END_IF
		END_IF

		MoversList[nMoverCount].nMoverIndex    := nMoverIndex; 
		MoversList[nMoverCount].nMoverPosition := nMoverPosition;
		MoversList[nMoverCount].nMoverTrackOID := nMoverTrackOID;
				
		
		sStatusMessage := CONCAT('AddMover: Success, added mover: ', UDINT_TO_STRING(nMoverIndex));
		nResult := 1;
	ELSE
		CASE nResult OF
		-11: sStatusMessage := 'AddMover: Invalid mover ID, Check P_Id';	
		-12: sStatusMessage := 'AddMover: Invalid track OID';
		-13: sStatusMessage := 'AddMover: Max number of movers in list exceeded.';
		-14: sStatusMessage := 'AddMover: Double entry, mover already in the list.';
		-15: sStatusMessage := 'AddMover: Empty mover interface';
		ELSE
			sStatusMessage := 'AddMover: Error';
		END_CASE		
	END_IF				
			
	AddMover := nResult;
	
	
	FOR idx:=10 TO 1 BY -1 DO 
		sHistoryAddMover[idx] := sHistoryAddMover[idx-1];
	END_FOR
	sText := CONCAT('Add Mover: ', UDINT_TO_STRING(nMoverIndex));
	sText := CONCAT(sText, ' Result: ');
	sText := CONCAT(sText, DINT_TO_STRING(nResult));
	sText := CONCAT(sText, ' ');
	sText := CONCAT(sText, sStatusMessage);
	sHistoryAddMover[0] := sText;
END_METHOD

METHOD AddTrack : DINT
VAR_INPUT
	i_Track	: I_TrackStandard;
END_VAR

VAR_INST	
	TrackInfo		: PlanarObjectInfo;
	nTrackOID		: UDINT;
	idx				: UDINT;
	nState	    	: INT;
	bDoubleEntry	: BOOL;

	nCycleTest		: UINT;
END_VAR



		nResult := 0;
		IF i_Track <> 0 THEN  		  
			TrackInfo := i_Track.P_Info;
			nTrackOID := TrackInfo.Id;
		END_IF
	
		
		// Check TrackOID
		IF nResult = 0 THEN
			IF nTrackOID > 0 THEN
				AddTrack := 0;
			ELSE
				nResult := -21;		
			END_IF
		END_IF
		
		
	    // Check for space
		IF nResult = 0 THEN 
			IF nTrackCount < maxTrackCount THEN
				nTrackCount := nTrackCount +1;	
			ELSE
				nResult := -22;
			END_IF	
		END_IF		
		
		
		// Check for double entry
		IF nResult = 0 THEN 
			bDoubleEntry := FALSE;
			FOR idx:=1 TO nTrackCount DO
				IF nTrackOIDs[idx] = nTrackOID THEN
					bDoubleEntry := TRUE;
				END_IF
			END_FOR
	
			IF bDoubleEntry THEN
				nResult := -23;		
			END_IF
		END_IF

		
	    // Adding Track
		IF nResult = 0 THEN 
			nTrackOIDs[nTrackCount] := nTrackOID;
			 TrackList[nTrackCount] := i_Track;
			 
			nResult := 1;
		END_IF
		
		
		
		
		
		
		IF nTrackCount = 1 THEN
			fLengthFirstTrack := i_Track.GetLength();
		END_IF
		
		
		
	    // Reult 
		CASE nResult OF
		  1: sStatusMessage := CONCAT('success: Added Track: ' , UDINT_TO_STRING(nTrackOID)); 
		-21: sStatusMessage := 'AddTrack: Invalid track OID.';	
	 	-22: sStatusMessage := 'AddTrack: Max number of tracks exceeded.';
		-23: sStatusMessage := 'AddTrack: Double entry, track already added.';
		ELSE
			sStatusMessage := 'Wrong input data';
		END_CASE		
		AddTrack := nResult;
END_METHOD

METHOD ClearList : BOOL
VAR_INPUT
END_VAR
VAR_INST
	nCycleTest	: INT;	
END_VAR
nCycleTest := nCycleTest + 1;

	   nResult := 0;	
sStatusMessage := 'List cleared';

nMoverCount := 0;
MEMSET(ADR(MoversList), 0, SIZEOF(MoversList));
MEMSET(ADR(MoversListITF), 0, SIZEOF(MoversListITF));
	
ClearList := TRUE;
END_METHOD

METHOD ClearTrackOrder : BOOL
VAR_INPUT
END_VAR





VAR_INST
	
	nCycleTest	: INT;
	idx			: UDINT;

END_VAR


	nCycleTest := nCycleTest +1;


		  nResult := 0;	
	sStatusMessage := 'Track order cleared';
	
	nTrackCount := 0;
	MEMSET(ADR(nTrackOIDs), 0, SIZEOF(nTrackOIDs));
	
	
	FOR idx:=1 TO maxTrackCount DO
		TrackList[idx] := 0;	
	END_FOR
	
	
	fSortingOrigin := 0.0;
	
	ClearTrackOrder := TRUE;
END_METHOD

{attribute 'hide'}
METHOD CopyList : I_List
VAR_INPUT
END_VAR




VAR_INST
	
	idx						: UDINT;
	nNumberOfMovers 		: UDINT;


END_VAR



	
	nNumberOfMovers := CopyList.P_nNumberInList;
	
	
	
	(*
	
	IF nNumberOfMovers > 0 THEN
		FOR idx:=1 TO nNumberOfMovers
			
		END_FOR
		
	*)
END_METHOD

METHOD GetMoverIndexInListPosition : UDINT
VAR_INPUT
	nListIndex	: UDINT;
END_VAR
	IF nMoverCount > 0 AND nListIndex <= nMoverCount THEN
		GetMoverIndexInListPosition := MoversList[nListIndex].nMoverIndex;
	ELSE
		GetMoverIndexInListPosition := 0;
	END_IF
END_METHOD

METHOD GetMoverInListPosition : I_XPlanarMoverStandard
VAR_INPUT
	nListPosition	: UDINT;
END_VAR
VAR
	idx				: UDINT;
END_VAR
GetMoverInListPosition := NoMover;

IF nMoverCount > 0 AND nListPosition <= nMoverCount AND nListPosition > 0 THEN
	FOR idx := 1 TO maxNumMover DO
		IF MoversListITF[idx] <> 0 AND_THEN MoversListITF[idx].P_Id = MoversList[nListPosition].nMoverIndex THEN
			GetMoverInListPosition := MoversListITF[idx];
			EXIT;
		END_IF
	END_FOR
END_IF
END_METHOD

PROPERTY P_FirstInList : I_XPlanarMoverStandard
GET
VAR
	
	idx	: UDINT;

END_VAR
P_FirstInList := NoMover;
IF nMoverCount > 0 AND MoversList[1].nMoverIndex > 0 THEN
	FOR idx := 1 TO maxNumMover DO
		IF MoversListITF[idx] <> 0 AND_THEN MoversListITF[idx].P_Id = MoversList[1].nMoverIndex THEN
			P_FirstInList := MoversListITF[idx];
			EXIT;
		END_IF
	END_FOR
END_IF
END_GET
END_PROPERTY

PROPERTY P_Message : STRING
GET
P_Message := sStatusMessage;
END_GET
END_PROPERTY

PROPERTY P_MoverList : REFERENCE TO ARRAY [1..maxNumMover] OF ST_MoverInList
GET
P_MoverList REF= MoversList;
END_GET
END_PROPERTY


PROPERTY P_NumberInList : UDINT
GET
   P_NumberInList := nMoverCount;
END_GET
END_PROPERTY

PROPERTY P_Result : DINT
GET

P_Result := nResult;
END_GET
END_PROPERTY

PROPERTY P_SortingDirection : eSortingDirection
GET


P_SortingDirection := nSortingDirection;
END_GET
SET

nSortingDirection := P_SortingDirection;
END_SET
END_PROPERTY

PROPERTY P_SortingOrigin : LREAL
GET
P_SortingOrigin := fSortingOrigin;
END_GET
SET

fSortingOrigin := P_SortingOrigin;
END_SET
END_PROPERTY

PROPERTY P_TrackBuiltInfo : ST_TrackBuiltInfo
GET
P_TrackBuiltInfo := TrackBuiltInfo;
END_GET
SET
TrackBuiltInfo := P_TrackBuiltInfo;
END_SET
END_PROPERTY

METHOD RemoveFirstInList : I_XPlanarMoverStandard
VAR_INPUT
END_VAR
VAR
	id				: UDINT;

	item			: UDINT;
	found			: BOOL;

	blockSize		: UDINT;
	movedItf		: UDINT;
	deletedItf		: UDINT;
	movedStruct		: UDINT;
	deletedStruct	: UDINT;

	idx				: UDINT;
END_VAR
RemoveFirstInList := NoMover;

nResult := 0;
sStatusMessage := '';

IF nMoverCount > 0 THEN
	idx := 1;
	id := MoversList[idx].nMoverIndex;

	found := FALSE;
	item := 1;
	WHILE item <= maxNumMover AND NOT found DO
		IF MoversListITF[item] = 0 THEN
			// Empty spot
			item := item + 1;
		ELSE
			// Check for matching mover ID
			found := MoversListITF[item].P_Id = id;
			IF NOT found THEN
				item := item + 1;
			END_IF
		END_IF
	END_WHILE

	IF NOT found THEN
		nResult := -12;
		sStatusMessage := 'RemoveFromList: Mover not found in list';
	END_IF

	IF nResult = 0 AND found THEN
		RemoveFirstInList := MoversListITF[item];

		// Shift the interfaces array content 1 position down, starting at found index
		blockSize := (maxNumMover - item) * SIZEOF(MoversListITF) / maxNumMover;
		IF blockSize > 0 THEN
			movedItf := MEMMOVE(destAddr:= ADR(MoversListITF[item]), srcAddr:= ADR(MoversListITF[item + 1]), n:= blockSize);
		END_IF
		deletedItf := MEMSET(destAddr:= ADR(MoversListITF[maxNumMover]), fillByte:= 0, n:= SIZEOF(MoversListITF) / maxNumMover);
	
		// Shift the structures array content 1 position down, starting at found index
		blockSize := (maxNumMover - idx) * SIZEOF(ST_MoverInList);
		IF blockSize > 0 THEN
			movedStruct := MEMMOVE(destAddr:= ADR(MoversList[idx]), srcAddr:= ADR(MoversList[idx + 1]), n:= blockSize);
		END_IF
		deletedStruct := MEMSET(destAddr:= ADR(MoversList[maxNumMover]), fillByte:= 0, n:= SIZEOF(ST_MoverInList));
				
		nMoverCount := nMoverCount - 1;
		
		nResult := 1;
		sStatusMessage := 'RemoveFirstInList: Success, mover removed';
	END_IF
ELSE
	nResult := -41;
	sStatusMessage := 'RemoveFirstInList: Mover list empty';			
END_IF

// Log operation
FOR idx := 10 TO 1 BY -1 DO 
	sHistoryAddMover[idx] := sHistoryAddMover[idx - 1];
END_FOR
sHistoryAddMover[0] := sStatusMessage;
END_METHOD

// Removes a mover from the list
METHOD RemoveFromList : DINT
VAR_INPUT
	ipMover			: I_XPlanarMoverStandard;	// Mover to remove
END_VAR
VAR
	id				: UDINT;

	item			: UDINT;
	found			: BOOL;

	blockSize		: UDINT;
	movedItf		: UDINT;
	deletedItf		: UDINT;
	movedStruct		: UDINT;
	deletedStruct	: UDINT;

	idx				: UDINT;

	sText			: STRING;
END_VAR
nResult := 0;
sStatusMessage := '';

IF ipMover = 0 THEN
	id := 0;
	nResult := -15;
	sStatusMessage := 'RemoveFromList: Empty mover interface';
END_IF

IF nResult = 0 THEN
	id := ipMover.P_Id;
	IF id = 0 THEN
		nResult := -11;
		sStatusMessage := 'RemoveFromList: Invalid mover ID, Check P_Id';
	END_IF
END_IF

IF nResult = 0 THEN
	found := FALSE;
	item := 1;
	WHILE item <= maxNumMover AND NOT found DO
		IF MoversListITF[item] = 0 THEN
			// Empty spot
			item := item + 1;
		ELSE
			// Check for matching mover ID
			found := MoversListITF[item].P_Id = id;
			IF NOT found THEN
				item := item + 1;
			END_IF
		END_IF
	END_WHILE
	
	IF found THEN
		// Mover found in ITF list, now search its position in struct list
		found := FALSE;
		idx := 1;
		WHILE idx <= maxNumMover AND NOT found DO
			IF MoversList[idx].nMoverIndex = 0 THEN
				// Empty spot
				idx := idx + 1;
			ELSE
				// Check for matching mover ID
				found := MoversList[idx].nMoverIndex = id;
				IF NOT found THEN
					idx := idx + 1;
				END_IF
			END_IF
		END_WHILE
	END_IF

	IF NOT found THEN
		nResult := -12;
		sStatusMessage := 'RemoveFromList: Mover not found in list';
	END_IF
END_IF

IF nResult = 0 AND found THEN
	// Shift the interfaces array content 1 position down, starting at found index
	blockSize := (maxNumMover - item) * SIZEOF(MoversListITF) / maxNumMover;
	IF blockSize > 0 THEN
		movedItf := MEMMOVE(destAddr:= ADR(MoversListITF[item]), srcAddr:= ADR(MoversListITF[item + 1]), n:= blockSize);
	END_IF
	deletedItf := MEMSET(destAddr:= ADR(MoversListITF[maxNumMover]), fillByte:= 0, n:= SIZEOF(MoversListITF) / maxNumMover);

	// Shift the structures array content 1 position down, starting at found index
	blockSize := (maxNumMover - idx) * SIZEOF(ST_MoverInList);
	IF blockSize > 0 THEN
		movedStruct := MEMMOVE(destAddr:= ADR(MoversList[idx]), srcAddr:= ADR(MoversList[idx + 1]), n:= blockSize);
	END_IF
	deletedStruct := MEMSET(destAddr:= ADR(MoversList[maxNumMover]), fillByte:= 0, n:= SIZEOF(ST_MoverInList));

	nMoverCount := nMoverCount - 1;

	nResult := 1;
	sStatusMessage := 'RemoveFromList: Success, mover removed';
END_IF

// Log operation
FOR idx := 10 TO 1 BY -1 DO
	sHistoryAddMover[idx] := sHistoryAddMover[idx - 1];
END_FOR
sText := CONCAT('Remove M', UDINT_TO_STRING(id));
sText := CONCAT(sText, ' from list. Result: ');
sText := CONCAT(sText, DINT_TO_STRING(nResult));
sText := CONCAT(sText, ' ');
sText := CONCAT(sText, sStatusMessage);
sHistoryAddMover[0] := sText;

// Return operation result
RemoveFromList := nResult;
END_METHOD

METHOD SortList : INT
VAR_INPUT
END_VAR



VAR_INST
	
	nState	    			: INT;	
	nTrackCounter			: UDINT;
	nSortingTrack			: UDINT;
	idx						: UDINT;
	idx1					: UDINT;
	idx2					: UDINT;
	nErrorID				: INT;
	fPositionHigh			: LREAL;
	nLastMover				: UDINT;
	MoversToSort			: ARRAY [1..maxNumMover] OF ST_MoverInList;
	MoversSorted			: ARRAY [1..maxNumMover] OF ST_MoverInList;
	nMoverSorted			: ARRAY [1..maxNumMover] OF BOOL;
	nMoverQueuCounter		: UDINT;
	nMoverQueuCounterTotal	: UDINT;
	nMoverLineDescending	: ARRAY [1..(maxTrackCount+1), 1..maxNumMover] OF UDINT;
	nMoverLineAscend		: ARRAY [1..maxNumMover] OF UDINT;
	nMoverLineDescend		: ARRAY [1..maxNumMover] OF UDINT;
	nMoverLineSorted		: ARRAY [1..maxNumMover] OF UDINT;
	nAscendingCounter		: UDINT;
	nDescendingCounter		: UDINT;
	nMoverLineCounter		: UDINT;	
	nListCounter			: UDINT;
	nTrackOID				: UDINT;
	nMoverInListIndex		: UDINT;
	bDoLoop					: BOOL;
	bTrackLineCheckOK		: BOOL;
	
	nMoverQueuCounterRemainTotal	: UDINT;
	
	sMoverSortedInfo				: STRING;
	
	thisSegment						: UDINT;	
	thisSegmentStartFromTrack		: UDINT;
	thisSegmentEndAtTrack			: UDINT;
	
	nextSegment						: UDINT;
	nextSegmentStartFromTrack		: UDINT;
	nextSegmentEndAtTrack			: UDINT;
	nFailedAt						: UDINT;	

	
END_VAR
 
	// Start
	nErrorID := 0;
	IF nErrorID = 0 THEN	
		IF nMoverCount > 0 THEN
			sStatusMessage := 'Sorting';
			 SortList := 0;
		ELSE
			nErrorID := -31;
		END_IF	
	END_IF
	
	
	// Check how many tracks to sort
	IF nErrorID = 0 THEN	
		nTrackCounter := 0;
		FOR idx:=1 TO maxTrackCount DO
			IF nTrackOIDs[idx] > 0 THEN 
				nTrackCounter := nTrackCounter +1;
			END_IF
		END_FOR
			
		IF nTrackCounter = 0 THEN
			nErrorID := -32;	
		END_IF	
	END_IF
	
	
	// Are all tracks in one line?
	        nFailedAt := 0;
	bTrackLineCheckOK := TRUE;
	FOR idx:=1 TO nTrackCounter DO
		IF idx < maxTrackCount THEN
			
			thisSegmentStartFromTrack := 0;
			    thisSegmentEndAtTrack := 0;
			nextSegmentStartFromTrack := 0;
			    nextSegmentEndAtTrack := 0;
					      nextSegment := 0;
						  
						  
			FOR idx2:=1 TO maxTrackCount DO
				IF TrackList[idx] <> 0 THEN	
					IF TrackList[idx].P_OID = TrackBuiltInfo.TrackInfo[idx2].TrackOID THEN
						thisSegment := TrackBuiltInfo.TrackInfo[idx2].TrackOID;
						IF TrackBuiltInfo.TrackInfo[idx2].StartFromTrack <> 0 THEN thisSegmentStartFromTrack := TrackBuiltInfo.TrackInfo[idx2].StartFromTrack.P_OID; END_IF			  
						IF TrackBuiltInfo.TrackInfo[idx2].EndAtTrack     <> 0 THEN     thisSegmentEndAtTrack := TrackBuiltInfo.TrackInfo[idx2].EndAtTrack.P_OID;     END_IF	  
						EXIT;	
					END_IF
				END_IF
			END_FOR
			
			FOR idx2:=1 TO maxTrackCount DO
				IF TrackList[idx+1] <> 0 THEN
					IF TrackList[idx+1].P_OID = TrackBuiltInfo.TrackInfo[idx2].TrackOID THEN
						nextSegment := TrackBuiltInfo.TrackInfo[idx2].TrackOID;
						IF TrackBuiltInfo.TrackInfo[idx2].StartFromTrack <> 0 THEN nextSegmentStartFromTrack := TrackBuiltInfo.TrackInfo[idx2].StartFromTrack.P_OID; END_IF			  
						IF TrackBuiltInfo.TrackInfo[idx2].EndAtTrack	 <> 0 THEN     nextSegmentEndAtTrack := TrackBuiltInfo.TrackInfo[idx2].EndAtTrack.P_OID;     END_IF	  
						EXIT;	
					END_IF
				END_IF
			END_FOR				
	
			IF nextSegment > 0 THEN
				IF nextSegment > 0 THEN				
					IF NOT (nextSegmentStartFromTrack = thisSegment) THEN
						IF NOT (thisSegmentEndAtTrack = nextSegment) THEN
							IF bTrackLineCheckOK THEN
								nFailedAt := idx;
							END_IF
							bTrackLineCheckOK := FALSE;
						END_IF
					END_IF
				END_IF
			END_IF

		END_IF
	END_FOR	
	
	IF NOT bTrackLineCheckOK THEN
		nErrorID := -36;
	END_IF

	
	
	
	IF nErrorID = 0 THEN
	
		// Preparing 
		          MoversToSort := MoversList;
		          nListCounter := 0;
	  	         nSortingTrack := 0;
		nMoverQueuCounterTotal := 0;
		           bTrackSplit := FALSE;
		MEMSET(ADR(nMoverSorted), 0, SIZEOF(nMoverSorted));
		MEMSET(ADR(nMoverLineDescending), 0, SIZEOF(nMoverLineDescending));
		
		
		// Updating MoverData
		FOR idx1:=1 TO nMoverCount DO
			FOR idx2:=1 TO maxNumMover DO
				IF MoversListITF[idx2] <> 0 THEN
					IF MoversToSort[idx1].nMoverIndex = MoversListITF[idx2].P_Id THEN
						MoversToSort[idx1].nMoverPosition := MoversListITF[idx2].P_SetOnTrack.SetPos;
						MoversToSort[idx1].nMoverTrackOID := MoversListITF[idx2].P_SetOnTrack.TrackOID;
						EXIT;
					END_IF		
				END_IF
			END_FOR
		END_FOR

		
		
		// Checking sorting point of origin
		IF fSortingOrigin >= fLengthFirstTrack THEN
			fSortingOrigin := 0.0;
			      nErrorID := -34;
		ELSIF fSortingOrigin < 0.0 THEN
			fSortingOrigin := 0.0;
			      nErrorID := -35;			
		END_IF
		
		
		// Sorting for all tracks		
		nMoverQueuCounter := 0;
		    nSortingTrack := 1;
			
		bDoLoop := TRUE;
		WHILE bDoLoop DO
			
			IF   nSortingTrack = 1 
			AND fSortingOrigin > 0.0 
			THEN
				  bTrackSplit := TRUE;
				fPositionHigh := fSortingOrigin;
			ELSE
				fPositionHigh := 0.0;
			END_IF				
		
			nLastMover := 0;
			FOR idx:=1 TO nMoverCount DO
				IF  MoversToSort[idx].nMoverTrackOID = nTrackOIDs[nSortingTrack] 
				AND MoversToSort[idx].nMoverPosition >= fPositionHigh
				AND NOT nMoverSorted[idx]
				THEN
					fPositionHigh := MoversToSort[idx].nMoverPosition;
					   nLastMover := idx;
				END_IF
			END_FOR
	
			IF nLastMover > 0 THEN	
					 nMoverQueuCounter := nMoverQueuCounter +1;
				nMoverQueuCounterTotal := nMoverQueuCounterTotal +1;
				nMoverLineDescending[nSortingTrack, nMoverQueuCounter] := MoversToSort[nLastMover].nMoverIndex; 
				nMoverSorted[nLastMover] := TRUE;
			ELSE
				nMoverQueuCounter := 0;
				nSortingTrack := nSortingTrack +1;
				IF nSortingTrack > nTrackCounter THEN
					bDoLoop := FALSE;	
				END_IF			
			END_IF
					
		END_WHILE
			
			
		
		IF bTrackSplit THEN	
			
			           nMoverQueuCounter := 0;
			nMoverQueuCounterRemainTotal := 0;
		
			bDoLoop := TRUE;
			WHILE bDoLoop DO
		
				fPositionHigh := 0.0;
				nSortingTrack := 1;
				   nLastMover := 0;
				   
				FOR idx:=1 TO nMoverCount DO
					IF  MoversToSort[idx].nMoverTrackOID = nTrackOIDs[nSortingTrack] 
					AND MoversToSort[idx].nMoverPosition >= fPositionHigh
					AND MoversToSort[idx].nMoverPosition < fSortingOrigin
					AND NOT nMoverSorted[idx]
					THEN
						fPositionHigh := MoversToSort[idx].nMoverPosition;
						   nLastMover := idx;
					END_IF
				END_FOR			
			
				IF nLastMover > 0 THEN	
							   nMoverQueuCounter := nMoverQueuCounter +1;
						  nMoverQueuCounterTotal := nMoverQueuCounterTotal +1;
					nMoverQueuCounterRemainTotal := nMoverQueuCounterRemainTotal +1;
					nMoverLineDescending[nTrackCounter+1, nMoverQueuCounter] := MoversToSort[nLastMover].nMoverIndex; 
					nMoverSorted[nLastMover] := TRUE;
				ELSE 
					bDoLoop := FALSE;
				END_IF			
			
			END_WHILE
		END_IF
			
		
		
				
	 	// Building the whole list 
		IF bTrackSplit THEN
	   		nListCounter := nTrackCounter +1;
		ELSE
			nListCounter := nTrackCounter;
		END_IF
		
		nMoverLineCounter := 0;
		WHILE (nListCounter > 0) DO
			
			IF nListCounter > nTrackCounter THEN
				nTrackOID := nTrackOIDs[1];
			ELSE 
				nTrackOID := nTrackOIDs[nListCounter];	
			END_IF
			
